C09104=1083.257,-6.050,442.174,174.206,19.488,153.253
C09105=1083.262,-5.800,442.160,174.207,19.490,153.253
C09106=1083.268,-5.551,442.147,174.208,19.492,153.254
C09107=1083.274,-5.301,442.133,174.210,19.495,153.254
C09108=1083.280,-5.052,442.120,174.212,19.496,153.254
C09109=1083.285,-4.803,442.106,174.213,19.498,153.254
C09110=1083.292,-4.553,442.092,174.214,19.500,153.254
C09111=1083.298,-4.303,442.078,174.216,19.503,153.254
C09112=1083.303,-4.053,442.064,174.218,19.504,153.254
C09113=1083.309,-3.804,442.051,174.219,19.506,153.254
C09114=1083.315,-3.555,442.037,174.220,19.508,153.255
C09115=1083.321,-3.305,442.024,174.222,19.510,153.255
C09116=1083.327,-3.055,442.010,174.224,19.512,153.255
C09117=1083.333,-2.805,441.996,174.225,19.514,153.255
C09118=1083.338,-2.556,441.982,174.226,19.516,153.255
C09119=1083.344,-2.307,441.969,174.228,19.519,153.255
C09120=1083.350,-2.057,441.955,174.229,19.521,153.255
C09121=1083.355,-1.807,441.941,174.231,19.523,153.256
C09122=1083.361,-1.558,441.927,174.232,19.524,153.256
C09123=1083.368,-1.282,441.912,174.234,19.527,153.256
C09124=1083.374,-1.007,441.897,174.235,19.529,153.256
C09125=1083.380,-0.732,441.882,174.237,19.532,153.256
C09126=1083.387,-0.457,441.866,174.238,19.534,153.256
C09127=1083.392,-0.207,441.852,174.241,19.536,153.256
C09128=1083.398,0.043,441.838,174.242,19.538,153.257
C09129=1083.403,0.292,441.824,174.243,19.540,153.257
C09130=1083.410,0.541,441.811,174.244,19.542,153.257
C09131=1083.416,0.792,441.796,174.247,19.545,153.257
C09132=1083.421,1.041,441.783,174.248,19.547,153.257
C09133=1083.427,1.290,441.768,174.249,19.548,153.257
C09134=1083.432,1.540,441.754,174.250,19.550,153.257
C09135=1083.439,1.789,441.741,174.253,19.553,153.258
C09136=1083.445,2.039,441.727,174.254,19.555,153.258
C09137=1083.450,2.289,441.713,174.255,19.557,153.258
C09138=1083.456,2.538,441.699,174.256,19.559,153.258
C09139=1083.461,2.787,441.684,174.259,19.561,153.258
C09140=1083.467,3.037,441.670,174.260,19.563,153.258
C09141=1083.474,3.287,441.657,174.261,19.565,153.258
C09142=1083.479,3.537,441.643,174.262,19.567,153.259
C09143=1083.485,3.785,441.628,174.264,19.569,153.259
C09144=1083.490,4.035,441.615,174.266,19.571,153.259
C09145=1083.496,4.285,441.600,174.267,19.573,153.259
C09146=1083.502,4.535,441.586,174.268,19.575,153.259
C09147=1083.508,4.784,441.572,174.270,19.577,153.259
C09148=1083.514,5.033,441.559,174.272,19.579,153.259
C09149=1083.520,5.283,441.544,174.273,19.581,153.260
C09150=1083.525,5.533,441.531,174.274,19.583,153.260
C09151=1083.531,5.782,441.516,174.276,19.585,153.260
C09152=1083.537,6.032,441.502,174.278,19.587,153.260
C09153=1083.543,6.282,441.488,174.279,19.589,153.260
C09154=1083.549,6.531,441.473,174.281,19.592,153.260
C09155=1083.554,6.780,441.459,174.282,19.594,153.261
C09156=1083.561,7.030,441.446,174.284,19.595,153.261
C09157=1083.567,7.279,441.431,174.285,19.597,153.261
C09158=1083.572,7.529,441.417,174.287,19.600,153.261
C09159=1083.578,7.778,441.403,174.288,19.602,153.261
C09160=1083.584,8.028,441.388,174.289,19.604,153.261
C09161=1083.589,8.278,441.375,174.291,19.606,153.261
C09162=1083.595,8.527,441.360,174.293,19.608,153.261
C09163=1083.601,8.777,441.346,174.294,19.610,153.262
C09164=1083.607,9.026,441.332,174.295,19.612,153.262
C09165=1083.613,9.275,441.317,174.298,19.615,153.262
C09166=1083.619,9.526,441.303,174.299,19.616,153.262
C09167=1083.625,9.774,441.289,174.300,19.618,153.262
C09168=1083.631,10.024,441.275,174.301,19.620,153.262
C09169=1083.637,10.274,441.260,174.304,19.623,153.262
C09170=1083.643,10.523,441.246,174.305,19.625,153.263
C09171=1083.649,10.773,441.232,174.306,19.626,153.263
C09172=1083.654,11.022,441.218,174.308,19.628,153.263
C09173=1083.660,11.272,441.204,174.310,19.631,153.263
C09174=1083.666,11.522,441.189,174.311,19.633,153.263
C09175=1083.672,11.771,441.175,174.312,19.635,153.263
C09176=1083.678,12.020,441.160,174.314,19.637,153.263
C09177=1083.684,12.270,441.146,174.316,19.639,153.263
C09178=1083.689,12.519,441.132,174.317,19.641,153.264
C09179=1083.695,12.770,441.117,174.318,19.643,153.264
C09180=1083.701,13.019,441.103,174.320,19.645,153.264
C09181=1083.707,13.268,441.089,174.322,19.647,153.264
C09182=1083.713,13.518,441.074,174.323,19.649,153.264
C09183=1083.719,13.767,441.059,174.325,19.651,153.264
C09184=1083.725,14.017,441.045,174.326,19.653,153.264
C09185=1083.731,14.266,441.031,174.328,19.655,153.265
C09186=1083.736,14.516,441.017,174.329,19.657,153.265
C09187=1083.744,14.793,441.000,174.331,19.659,153.265
C09188=1083.749,15.071,440.984,174.332,19.661,153.265
C09189=1083.756,15.348,440.968,174.334,19.664,153.265
C09190=1083.763,15.625,440.952,174.336,19.666,153.265
C09191=1083.768,15.874,440.937,174.338,19.668,153.265
C09192=1083.774,16.125,440.923,174.339,19.670,153.266
C09193=1083.780,16.373,440.908,174.340,19.672,153.266
C09194=1083.786,16.623,440.894,174.342,19.675,153.266
C09195=1083.791,16.873,440.880,174.344,19.676,153.266
C09196=1083.797,17.122,440.865,174.345,19.678,153.266
C09197=1083.803,17.372,440.850,174.347,19.681,153.266
C09198=1083.808,17.621,440.836,174.348,19.683,153.267
C09199=1083.815,17.871,440.821,174.350,19.685,153.267
C09200=1083.820,18.120,440.806,174.352,19.687,153.267
C09201=1083.827,18.370,440.792,174.353,19.689,153.267
C09202=1083.832,18.619,440.777,174.354,19.691,153.267
C09203=1083.837,18.868,440.762,174.356,19.693,153.267
C09204=1083.844,19.118,440.747,174.358,19.695,153.267
C09205=1083.849,19.368,440.733,174.359,19.697,153.268
C09206=1083.856,19.617,440.718,174.360,19.699,153.268
C09207=1083.861,19.866,440.704,174.362,19.701,153.268
C09208=1083.867,20.117,440.689,174.364,19.703,153.268
C09209=1083.872,20.366,440.674,174.365,19.706,153.268
C09210=1083.879,20.615,440.659,174.367,19.708,153.268
C09211=1083.885,20.864,440.645,174.368,19.710,153.268
C09212=1083.889,21.114,440.630,174.370,19.712,153.268
C09213=1083.896,21.364,440.615,174.371,19.714,153.269
C09214=1083.902,21.613,440.601,174.373,19.716,153.269
C09215=1083.907,21.863,440.585,174.374,19.718,153.269
C09216=1083.913,22.112,440.571,174.376,19.720,153.269
C09217=1083.919,22.362,440.557,174.378,19.723,153.269
C09218=1083.924,22.611,440.541,174.379,19.725,153.269
C09219=1083.930,22.861,440.526,174.380,19.726,153.269
C09220=1083.936,23.110,440.512,174.382,19.729,153.270
C09221=1083.942,23.360,440.496,174.384,19.731,153.270
C09222=1083.948,23.609,440.482,174.385,19.733,153.270
C09223=1083.954,23.859,440.467,174.387,19.735,153.270
C09224=1083.959,24.108,440.452,174.389,19.737,153.270
C09225=1083.965,24.358,440.437,174.390,19.739,153.270
C09226=1083.971,24.607,440.423,174.392,19.741,153.270
C09227=1083.977,24.857,440.407,174.393,19.743,153.271
C09228=1083.982,25.106,440.393,174.394,19.745,153.271
C09229=1083.989,25.356,440.378,174.396,19.748,153.271
C09230=1083.994,25.605,440.363,174.398,19.749,153.271
C09231=1084.000,25.854,440.348,174.399,19.751,153.271
C09232=1084.006,26.103,440.333,174.400,19.753,153.271
C09233=1084.012,26.353,440.317,174.403,19.756,153.271
C09234=1084.017,26.603,440.304,174.404,19.758,153.272
C09235=1084.024,26.853,440.289,174.405,19.759,153.272
C09236=1084.029,27.102,440.274,174.407,19.762,153.272
C09237=1084.035,27.352,440.259,174.409,19.764,153.272
C09238=1084.040,27.601,440.243,174.410,19.766,153.272
C09239=1084.046,27.850,440.228,174.412,19.768,153.272
C09240=1084.052,28.100,440.213,174.413,19.770,153.272
C09241=1084.058,28.349,440.198,174.415,19.772,153.273
C09242=1084.064,28.599,440.183,174.417,19.774,153.273
C09243=1084.069,28.848,440.168,174.418,19.776,153.273
C09244=1084.076,29.098,440.153,174.419,19.778,153.273
C09245=1084.081,29.347,440.138,174.422,19.780,153.273
C09246=1084.087,29.597,440.123,174.423,19.782,153.273
C09247=1084.092,29.846,440.108,174.424,19.784,153.273
C09248=1084.098,30.096,440.093,174.426,19.787,153.274
C09249=1084.104,30.345,440.077,174.427,19.789,153.274
C09250=1084.109,30.594,440.062,174.429,19.791,153.274
C09251=1084.116,30.874,440.045,174.431,19.793,153.274
C09252=1084.123,31.152,440.028,174.433,19.796,153.274
C09253=1084.128,31.431,440.011,174.434,19.798,153.274
C09254=1084.135,31.710,439.995,174.436,19.800,153.275
C09255=1084.141,31.959,439.978,174.437,19.802,153.275
C09256=1084.147,32.208,439.964,174.440,19.804,153.275
C09257=1084.153,32.458,439.948,174.441,19.806,153.275
C09258=1084.158,32.707,439.934,174.442,19.808,153.275
C09259=1084.164,32.957,439.918,174.444,19.811,153.275
C09260=1084.170,33.207,439.903,174.446,19.813,153.275
C09261=1084.176,33.456,439.888,174.447,19.814,153.275
C09262=1084.181,33.705,439.872,174.449,19.817,153.276
C09263=1084.187,33.954,439.857,174.450,19.819,153.276
C09264=1084.193,34.204,439.842,174.452,19.821,153.276
C09265=1084.199,34.454,439.827,174.454,19.823,153.276
C09266=1084.204,34.703,439.811,174.455,19.825,153.276
C09267=1084.211,34.952,439.796,174.456,19.827,153.276
C09268=1084.217,35.202,439.780,174.459,19.829,153.276
C09269=1084.222,35.451,439.765,174.460,19.831,153.277
C09270=1084.228,35.701,439.750,174.461,19.833,153.277
C09271=1084.234,35.951,439.735,174.463,19.835,153.277
C09272=1084.239,36.200,439.719,174.465,19.837,153.277
C09273=1084.245,36.449,439.704,174.466,19.839,153.277
C09274=1084.251,36.699,439.688,174.468,19.842,153.277
C09275=1084.257,36.948,439.673,174.469,19.843,153.277
C09276=1084.263,37.198,439.657,174.471,19.845,153.277
C09277=1084.268,37.448,439.642,174.473,19.848,153.278
C09278=1084.274,37.697,439.627,174.474,19.850,153.278
C09279=1084.280,37.946,439.611,174.476,19.852,153.278
C09280=1084.286,38.196,439.595,174.478,19.854,153.278
C09281=1084.291,38.445,439.580,174.479,19.856,153.278
C09282=1084.298,38.694,439.565,174.481,19.858,153.278
C09283=1084.303,38.944,439.549,174.482,19.860,153.278
C09284=1084.308,39.193,439.534,174.484,19.862,153.279
C09285=1084.314,39.443,439.518,174.486,19.864,153.279
C09286=1084.321,39.692,439.503,174.487,19.866,153.279
C09287=1084.326,39.942,439.487,174.488,19.868,153.279
C09288=1084.332,40.191,439.471,174.490,19.871,153.279
C09289=1084.337,40.441,439.456,174.492,19.872,153.279
C09290=1084.343,40.690,439.440,174.494,19.875,153.279
C09291=1084.349,40.939,439.425,174.495,19.877,153.280
C09292=1084.355,41.189,439.409,174.497,19.879,153.280
C09293=1084.360,41.438,439.393,174.499,19.881,153.280
C09294=1084.366,41.688,439.378,174.500,19.883,153.280
C09295=1084.372,41.937,439.362,174.501,19.885,153.280
C09296=1084.378,42.187,439.347,174.503,19.887,153.280
C09297=1084.383,42.436,439.331,174.505,19.889,153.280
C09298=1084.389,42.686,439.315,174.506,19.891,153.280
C09299=1084.395,42.936,439.300,174.508,19.893,153.281
C09300=1084.400,43.184,439.284,174.510,19.895,153.281
C09301=1084.406,43.434,439.268,174.512,19.898,153.281
C09302=1084.412,43.683,439.253,174.513,19.899,153.281
C09303=1084.418,43.933,439.237,174.514,19.901,153.281
C09304=1084.423,44.182,439.221,174.516,19.904,153.281
C09305=1084.429,44.432,439.206,174.518,19.906,153.281
C09306=1084.435,44.681,439.189,174.519,19.908,153.282
C09307=1084.440,44.930,439.174,174.521,19.910,153.282
C09308=1084.446,45.180,439.158,174.523,19.912,153.282
C09309=1084.452,45.430,439.142,174.525,19.914,153.282
C09310=1084.457,45.679,439.126,174.526,19.916,153.282
C09311=1084.463,45.928,439.110,174.527,19.918,153.282
C09312=1084.468,46.178,439.095,174.529,19.921,153.282
C09313=1084.474,46.427,439.078,174.531,19.922,153.282
C09314=1084.479,46.677,439.062,174.533,19.925,153.283
C09315=1084.486,46.955,439.045,174.534,19.927,153.283
C09316=1084.492,47.234,439.027,174.536,19.929,153.283
C09317=1084.499,47.513,439.010,174.538,19.932,153.283
C09318=1084.505,47.791,438.992,174.540,19.934,153.283
C09319=1084.511,48.041,438.976,174.542,19.936,153.283
C09320=1084.516,48.291,438.960,174.543,19.938,153.284
C09321=1084.522,48.540,438.944,174.544,19.940,153.284
C09322=1084.527,48.789,438.928,174.547,19.942,153.284
C09323=1084.533,49.039,438.912,174.548,19.944,153.284
C09324=1084.538,49.288,438.896,174.550,19.946,153.284
C09325=1084.544,49.538,438.879,174.551,19.948,153.284
C09326=1084.550,49.788,438.864,174.553,19.950,153.284
C09327=1084.555,50.036,438.848,174.555,19.952,153.284
C09328=1084.561,50.286,438.832,174.556,19.954,153.285
C09329=1084.567,50.535,438.815,174.558,19.956,153.285
C09330=1084.573,50.785,438.800,174.560,19.958,153.285
C09331=1084.579,51.034,438.784,174.561,19.960,153.285
C09332=1084.584,51.283,438.768,174.563,19.963,153.285
C09333=1084.590,51.533,438.752,174.564,19.964,153.285
C09334=1084.596,51.782,438.736,174.567,19.967,153.285
C09335=1084.602,52.032,438.720,174.568,19.969,153.285
C09336=1084.607,52.281,438.703,174.569,19.971,153.286
C09337=1084.613,52.531,438.687,174.571,19.973,153.286
C09338=1084.618,52.780,438.671,174.573,19.975,153.286
C09339=1084.624,53.029,438.655,174.575,19.977,153.286
C09340=1084.630,53.279,438.639,174.576,19.979,153.286
C09341=1084.636,53.528,438.623,174.577,19.981,153.286
C09342=1084.641,53.778,438.607,174.580,19.983,153.286
C09343=1084.647,54.027,438.591,174.581,19.985,153.286
C09344=1084.653,54.277,438.574,174.583,19.987,153.287
C09345=1084.659,54.526,438.558,174.584,19.989,153.287
C09346=1084.664,54.775,438.542,174.586,19.991,153.287
C09347=1084.670,55.024,438.526,174.588,19.993,153.287
C09348=1084.676,55.274,438.509,174.589,19.995,153.287
C09349=1084.681,55.524,438.494,174.592,19.997,153.287
C09350=1084.687,55.773,438.477,174.593,19.999,153.287
C09351=1084.693,56.023,438.461,174.594,20.001,153.287
C09352=1084.699,56.272,438.444,174.597,20.003,153.287
C09353=1084.704,56.521,438.428,174.598,20.005,153.288
C09354=1084.710,56.771,438.412,174.600,20.008,153.288
C09355=1084.716,57.020,438.396,174.601,20.009,153.288
C09356=1084.722,57.269,438.379,174.603,20.011,153.288
C09357=1084.728,57.519,438.362,174.605,20.014,153.288
C09358=1084.733,57.768,438.346,174.606,20.015,153.288
C09359=1084.739,58.017,438.330,174.608,20.018,153.288
C09360=1084.745,58.266,438.314,174.610,20.019,153.288
C09361=1084.751,58.516,438.298,174.612,20.022,153.289
C09362=1084.757,58.765,438.282,174.613,20.024,153.289
C09363=1084.762,59.015,438.265,174.615,20.025,153.289
C09364=1084.768,59.264,438.248,174.617,20.028,153.289
C09365=1084.774,59.513,438.232,174.618,20.029,153.289
C09366=1084.780,59.763,438.216,174.620,20.031,153.289
C09367=1084.786,60.012,438.200,174.622,20.033,153.289
C09368=1084.791,60.262,438.183,174.624,20.035,153.289
C09369=1084.797,60.511,438.167,174.625,20.037,153.289
C09370=1084.803,60.761,438.150,174.627,20.039,153.289
C09371=1084.809,61.010,438.134,174.629,20.041,153.290
C09372=1084.814,61.260,438.117,174.630,20.043,153.290
C09373=1084.820,61.509,438.101,174.632,20.045,153.290
C09374=1084.826,61.758,438.085,174.634,20.047,153.290
C09375=1084.832,62.008,438.068,174.635,20.049,153.290
C09376=1084.838,62.257,438.052,174.637,20.051,153.290
C09377=1084.843,62.507,438.035,174.639,20.053,153.290
C09378=1084.850,62.757,438.019,174.641,20.055,153.290
C09379=1084.856,63.034,438.000,174.642,20.057,153.290
C09380=1084.862,63.313,437.982,174.644,20.059,153.291
C09381=1084.869,63.591,437.963,174.647,20.062,153.291
C09382=1084.876,63.870,437.945,174.649,20.064,153.291
C09383=1084.881,64.120,437.928,174.650,20.066,153.291
C09384=1084.887,64.369,437.912,174.652,20.068,153.291
C09385=1084.893,64.618,437.895,174.654,20.070,153.291
C09386=1084.898,64.867,437.878,174.655,20.072,153.291
C09387=1084.904,65.117,437.862,174.657,20.074,153.291
C09388=1084.909,65.366,437.845,174.659,20.076,153.291
C09389=1084.916,65.616,437.829,174.661,20.078,153.292
C09390=1084.922,65.865,437.812,174.662,20.080,153.292
C09391=1084.927,66.115,437.795,174.664,20.082,153.292
C09392=1084.933,66.364,437.778,174.666,20.084,153.292
C09393=1084.939,66.614,437.762,174.667,20.086,153.292
C09394=1084.945,66.863,437.745,174.669,20.087,153.292
C09395=1084.950,67.112,437.728,174.671,20.089,153.292
C09396=1084.956,67.362,437.712,174.673,20.092,153.292
C09397=1084.961,67.611,437.695,174.674,20.093,153.292
C09398=1084.967,67.860,437.678,174.676,20.096,153.292
C09399=1084.973,68.110,437.661,174.678,20.097,153.293
C09400=1084.979,68.359,437.645,174.680,20.100,153.293
C09401=1084.984,68.608,437.627,174.682,20.101,153.293
C09402=1084.990,68.857,437.611,174.684,20.104,153.293
C09403=1084.995,69.107,437.594,174.685,20.105,153.293
C09404=1085.002,69.356,437.577,174.686,20.107,153.293
C09405=1085.007,69.606,437.560,174.689,20.109,153.293
C09406=1085.013,69.855,437.543,174.690,20.111,153.293
C09407=1085.019,70.105,437.526,174.692,20.114,153.293
C09408=1085.025,70.354,437.510,174.694,20.115,153.293
C09409=1085.030,70.604,437.493,174.696,20.118,153.294
C09410=1085.036,70.853,437.475,174.697,20.119,153.294
C09411=1085.042,71.102,437.459,174.699,20.122,153.294
C09412=1085.047,71.352,437.442,174.701,20.123,153.294
C09413=1085.053,71.600,437.425,174.703,20.126,153.294
C09414=1085.058,71.850,437.408,174.704,20.127,153.294
C09415=1085.064,72.099,437.391,174.706,20.129,153.294
C09416=1085.070,72.349,437.374,174.708,20.131,153.294
C09417=1085.076,72.598,437.357,174.709,20.133,153.294
C09418=1085.081,72.848,437.340,174.712,20.135,153.294
C09419=1085.087,73.097,437.323,174.713,20.137,153.295
C09420=1085.092,73.346,437.306,174.715,20.139,153.295
C09421=1085.098,73.596,437.289,174.717,20.141,153.295
C09422=1085.104,73.845,437.272,174.719,20.143,153.295
C09423=1085.109,74.094,437.255,174.720,20.145,153.295
C09424=1085.115,74.344,437.237,174.722,20.147,153.295
C09425=1085.121,74.593,437.221,174.724,20.149,153.295
C09426=1085.127,74.842,437.203,174.726,20.151,153.295
C09427=1085.132,75.092,437.187,174.727,20.153,153.295
C09428=1085.138,75.341,437.170,174.730,20.155,153.295
C09429=1085.144,75.590,437.152,174.731,20.157,153.295
C09430=1085.150,75.840,437.135,174.733,20.159,153.295
C09431=1085.155,76.089,437.117,174.735,20.161,153.296
C09432=1085.161,76.339,437.101,174.737,20.163,153.296
C09433=1085.167,76.588,437.083,174.738,20.165,153.296
C09434=1085.172,76.837,437.067,174.740,20.166,153.296
C09435=1085.179,77.087,437.049,174.742,20.169,153.296
C09436=1085.184,77.336,437.032,174.743,20.170,153.296
C09437=1085.189,77.585,437.015,174.745,20.173,153.296
C09438=1085.195,77.834,436.997,174.747,20.174,153.296
C09439=1085.201,78.084,436.981,174.749,20.176,153.296
C09440=1085.207,78.333,436.963,174.751,20.178,153.296
C09441=1085.212,78.583,436.946,174.753,20.180,153.296
C09442=1085.218,78.832,436.929,174.754,20.182,153.297
C09443=1085.224,79.110,436.910,174.757,20.184,153.297
C09444=1085.231,79.389,436.890,174.759,20.186,153.297
C09445=1085.237,79.667,436.870,174.761,20.189,153.297
C09446=1085.243,79.945,436.851,174.762,20.190,153.297
C09447=1085.248,80.195,436.834,174.764,20.193,153.297
C09448=1085.254,80.445,436.816,174.766,20.194,153.297
C09449=1085.260,80.694,436.799,174.768,20.197,153.297
C09450=1085.266,80.943,436.782,174.769,20.198,153.297
C09451=1085.271,81.192,436.765,174.772,20.201,153.297
C09452=1085.277,81.441,436.747,174.773,20.202,153.298
C09453=1085.283,81.691,436.729,174.775,20.205,153.298
C09454=1085.288,81.941,436.712,174.777,20.206,153.298
C09455=1085.294,82.190,436.695,174.779,20.208,153.298
C09456=1085.299,82.439,436.677,174.780,20.210,153.298
C09457=1085.305,82.688,436.659,174.783,20.212,153.298
C09458=1085.311,82.937,436.642,174.784,20.214,153.298
C09459=1085.316,83.187,436.625,174.786,20.216,153.298
C09460=1085.322,83.436,436.607,174.788,20.218,153.298
C09461=1085.328,83.686,436.589,174.790,20.220,153.298
C09462=1085.333,83.935,436.572,174.791,20.221,153.298
C09463=1085.339,84.184,436.554,174.794,20.224,153.298
C09464=1085.344,84.434,436.537,174.795,20.225,153.299
C09465=1085.350,84.683,436.519,174.797,20.228,153.299
C09466=1085.356,84.932,436.502,174.799,20.229,153.299
C09467=1085.361,85.181,436.484,174.801,20.231,153.299
C09468=1085.367,85.431,436.466,174.802,20.233,153.299
C09469=1085.373,85.680,436.449,174.805,20.235,153.299
C09470=1085.379,85.929,436.432,174.807,20.237,153.299
C09471=1085.385,86.179,436.414,174.808,20.239,153.299
C09472=1085.391,86.428,436.396,174.811,20.241,153.299
C09473=1085.396,86.677,436.379,174.812,20.242,153.299
C09474=1085.402,86.927,436.362,174.814,20.245,153.299
C09475=1085.408,87.176,436.344,174.816,20.246,153.299
C09476=1085.413,87.425,436.326,174.818,20.248,153.299
C09477=1085.419,87.675,436.308,174.819,20.250,153.300
C09478=1085.425,87.924,436.291,174.822,20.252,153.300
C09479=1085.430,88.173,436.273,174.823,20.254,153.300
C09480=1085.436,88.423,436.255,174.825,20.256,153.300
C09481=1085.442,88.672,436.238,174.827,20.258,153.300
C09482=1085.447,88.921,436.220,174.829,20.260,153.300
C09483=1085.453,89.171,436.202,174.831,20.261,153.300
C09484=1085.458,89.420,436.184,174.833,20.264,153.300
C09485=1085.464,89.669,436.167,174.834,20.265,153.300
C09486=1085.470,89.919,436.149,174.837,20.267,153.300
C09487=1085.475,90.168,436.131,174.838,20.269,153.300
C09488=1085.482,90.418,436.113,174.840,20.271,153.300
C09489=1085.487,90.667,436.096,174.842,20.272,153.300
C09490=1085.493,90.916,436.077,174.844,20.274,153.300
C09491=1085.499,91.165,436.059,174.845,20.276,153.300
C09492=1085.504,91.414,436.042,174.848,20.278,153.300
C09493=1085.511,91.663,436.024,174.850,20.280,153.300
C09494=1085.515,91.913,436.006,174.851,20.282,153.301
C09495=1085.521,92.162,435.988,174.854,20.284,153.301
C09496=1085.527,92.412,435.970,174.855,20.286,153.301
C09497=1085.533,92.661,435.953,174.857,20.288,153.301
C09498=1085.537,92.910,435.935,174.859,20.290,153.301
C09499=1085.544,93.159,435.916,174.861,20.292,153.301
C09500=1085.549,93.408,435.898,174.863,20.293,153.301
C09501=1085.555,93.658,435.880,174.865,20.296,153.301
C09502=1085.560,93.907,435.862,174.866,20.297,153.301
C09503=1085.566,94.156,435.845,174.869,20.299,153.301
C09504=1085.572,94.406,435.827,174.870,20.301,153.301
C09505=1085.578,94.654,435.808,174.872,20.303,153.301
C09506=1085.583,94.905,435.790,174.875,20.305,153.301
C09507=1085.589,95.183,435.770,174.876,20.306,153.301
C09508=1085.595,95.461,435.750,174.878,20.309,153.302
C09509=1085.602,95.740,435.730,174.881,20.311,153.302
C09510=1085.608,96.018,435.710,174.883,20.313,153.302
C09511=1085.614,96.267,435.691,174.885,20.315,153.302
C09512=1085.620,96.517,435.674,174.887,20.317,153.302
C09513=1085.625,96.767,435.655,174.889,20.319,153.302
C09514=1085.631,97.016,435.637,174.890,20.321,153.302
C09515=1085.637,97.265,435.619,174.893,20.323,153.302
C09516=1085.643,97.514,435.601,174.894,20.324,153.302
C09517=1085.647,97.763,435.583,174.896,20.326,153.302
C09518=1085.654,98.012,435.564,174.898,20.327,153.302
C09519=1085.659,98.261,435.547,174.900,20.329,153.302
C09520=1085.665,98.511,435.528,174.902,20.332,153.302
C09521=1085.671,98.760,435.510,174.904,20.333,153.302
C09522=1085.677,99.010,435.492,174.906,20.335,153.302
C09523=1085.681,99.259,435.474,174.908,20.337,153.302
C09524=1085.688,99.508,435.455,174.910,20.339,153.302
C09525=1085.693,99.757,435.438,174.912,20.340,153.302
C09526=1085.699,100.006,435.419,174.914,20.343,153.302
C09527=1085.705,100.256,435.401,174.915,20.344,153.303
C09528=1085.711,100.505,435.383,174.918,20.346,153.303
C09529=1085.716,100.755,435.364,174.920,20.348,153.303
C09530=1085.722,101.004,435.346,174.921,20.349,153.303
C09531=1085.728,101.253,435.328,174.924,20.351,153.303
C09532=1085.733,101.502,435.309,174.925,20.353,153.303
C09533=1085.740,101.751,435.291,174.927,20.355,153.303
C09534=1085.744,102.001,435.273,174.929,20.357,153.303
C09535=1085.750,102.250,435.255,174.931,20.359,153.303
C09536=1085.756,102.499,435.236,174.934,20.361,153.303
C09537=1085.761,102.749,435.217,174.935,20.362,153.303
C09538=1085.767,102.998,435.199,174.937,20.365,153.303
C09539=1085.772,103.248,435.180,174.939,20.366,153.303
C09540=1085.778,103.496,435.162,174.941,20.368,153.303
C09541=1085.783,103.746,435.144,174.943,20.370,153.303
C09542=1085.789,103.995,435.125,174.945,20.371,153.303
C09543=1085.795,104.244,435.106,174.947,20.373,153.303
C09544=1085.800,104.493,435.089,174.949,20.375,153.303
C09545=1085.806,104.742,435.069,174.951,20.377,153.303
C09546=1085.812,104.992,435.051,174.952,20.379,153.303
C09547=1085.817,105.241,435.033,174.955,20.381,153.303
C09548=1085.823,105.491,435.014,174.957,20.383,153.303
C09549=1085.828,105.739,434.996,174.959,20.384,153.303
C09550=1085.834,105.989,434.976,174.961,20.386,153.303
C09551=1085.840,106.238,434.959,174.963,20.388,153.303
C09552=1085.845,106.487,434.940,174.965,20.390,153.303
C09553=1085.851,106.737,434.922,174.967,20.392,153.303
C09554=1085.857,106.986,434.903,174.969,20.393,153.304
C09555=1085.862,107.235,434.884,174.971,20.395,153.304
C09556=1085.868,107.484,434.866,174.972,20.397,153.304
C09557=1085.873,107.734,434.847,174.975,20.399,153.304
C09558=1085.880,107.983,434.828,174.977,20.401,153.304
C09559=1085.885,108.232,434.810,174.979,20.402,153.304
C09560=1085.890,108.482,434.791,174.981,20.404,153.304
C09561=1085.897,108.731,434.772,174.982,20.406,153.304
C09562=1085.902,108.979,434.753,174.985,20.408,153.304
C09563=1085.908,109.229,434.735,174.987,20.410,153.304
C09564=1085.913,109.478,434.716,174.989,20.411,153.304
C09565=1085.919,109.727,434.697,174.991,20.413,153.304
C09566=1085.925,109.976,434.678,174.993,20.414,153.304
C09567=1085.930,110.226,434.660,174.995,20.416,153.304
C09568=1085.936,110.475,434.641,174.997,20.418,153.304
C09569=1085.942,110.724,434.622,174.999,20.420,153.304
C09570=1085.948,110.974,434.603,175.001,20.422,153.304
C09571=1085.953,111.252,434.582,175.003,20.424,153.304
C09572=1085.960,111.531,434.562,175.006,20.426,153.304
C09573=1085.967,111.810,434.541,175.008,20.428,153.304
C09574=1085.973,112.088,434.520,175.010,20.429,153.304
C09575=1085.978,112.337,434.501,175.012,20.431,153.304
C09576=1085.984,112.586,434.482,175.014,20.433,153.304
C09577=1085.990,112.836,434.463,175.016,20.434,153.304
C09578=1085.995,113.084,434.444,175.018,20.436,153.304
C09579=1086.001,113.334,434.425,175.021,20.438,153.304
C09580=1086.007,113.583,434.406,175.022,20.440,153.304
C09581=1086.012,113.832,434.387,175.025,20.442,153.304
C09582=1086.018,114.082,434.369,175.026,20.443,153.304
C09583=1086.023,114.331,434.350,175.028,20.445,153.304
C09584=1086.029,114.580,434.331,175.031,20.447,153.304
C09585=1086.034,114.829,434.311,175.032,20.449,153.304
C09586=1086.040,115.079,434.292,175.035,20.451,153.304
C09587=1086.045,115.328,434.273,175.037,20.452,153.304
C09588=1086.051,115.577,434.255,175.038,20.454,153.304
C09589=1086.057,115.826,434.235,175.041,20.456,153.305
C09590=1086.062,116.075,434.217,175.042,20.458,153.305
C09591=1086.068,116.324,434.197,175.044,20.460,153.305
C09592=1086.074,116.574,434.178,175.047,20.462,153.305
C09593=1086.079,116.823,434.159,175.048,20.463,153.305
C09594=1086.084,117.072,434.140,175.051,20.465,153.305
C09595=1086.090,117.321,434.121,175.053,20.467,153.305
C09596=1086.096,117.571,434.101,175.055,20.469,153.305
C09597=1086.101,117.819,434.083,175.057,20.471,153.305
C09598=1086.106,118.069,434.063,175.059,20.472,153.305
C09599=1086.112,118.318,434.044,175.061,20.473,153.305
C09600=1086.118,118.568,434.025,175.063,20.475,153.305
C09601=1086.123,118.817,434.006,175.066,20.477,153.305
C09602=1086.129,119.066,433.987,175.067,20.479,153.305
C09603=1086.134,119.315,433.968,175.070,20.481,153.305
C09604=1086.140,119.564,433.948,175.071,20.482,153.305
C09605=1086.145,119.813,433.929,175.073,20.484,153.305
C09606=1086.151,120.062,433.909,175.076,20.486,153.305
C09607=1086.157,120.312,433.890,175.077,20.488,153.305
C09608=1086.162,120.561,433.871,175.080,20.489,153.305
C09609=1086.168,120.810,433.852,175.082,20.491,153.305
C09610=1086.173,121.059,433.833,175.084,20.493,153.305
C09611=1086.179,121.308,433.813,175.086,20.495,153.305
C09612=1086.185,121.558,433.794,175.088,20.497,153.305
C09613=1086.191,121.807,433.774,175.090,20.498,153.305
C09614=1086.196,122.056,433.755,175.092,20.500,153.305
C09615=1086.201,122.305,433.736,175.095,20.502,153.305
C09616=1086.207,122.555,433.717,175.096,20.503,153.305
C09617=1086.212,122.804,433.696,175.099,20.505,153.305
C09618=1086.218,123.053,433.677,175.101,20.507,153.305
C09619=1086.223,123.302,433.658,175.102,20.508,153.305
C09620=1086.229,123.551,433.639,175.105,20.510,153.305
C09621=1086.235,123.800,433.619,175.107,20.512,153.305
C09622=1086.240,124.050,433.600,175.109,20.513,153.305
C09623=1086.246,124.299,433.581,175.111,20.515,153.305
C09624=1086.252,124.548,433.561,175.114,20.517,153.305
C09625=1086.258,124.797,433.541,175.115,20.519,153.305
C09626=1086.263,125.046,433.523,175.118,20.520,153.305
C09627=1086.269,125.295,433.503,175.120,20.522,153.305
C09628=1086.275,125.544,433.483,175.122,20.523,153.305
C09629=1086.280,125.794,433.464,175.124,20.525,153.305
C09630=1086.286,126.043,433.444,175.127,20.527,153.305
C09631=1086.291,126.292,433.424,175.128,20.528,153.305
C09632=1086.297,126.542,433.405,175.130,20.530,153.305
C09633=1086.303,126.791,433.385,175.133,20.532,153.305
C09634=1086.309,127.040,433.366,175.134,20.533,153.305
C09635=1086.315,127.318,433.344,175.137,20.535,153.305
C09636=1086.321,127.597,433.322,175.139,20.537,153.305
C09637=1086.328,127.875,433.300,175.142,20.539,153.305
C09638=1086.334,128.154,433.279,175.144,20.541,153.305
C09639=1086.340,128.403,433.259,175.147,20.542,153.305
C09640=1086.345,128.652,433.240,175.149,20.544,153.305
C09641=1086.351,128.901,433.219,175.151,20.546,153.305
C09642=1086.356,129.151,433.200,175.153,20.548,153.305
C09643=1086.362,129.400,433.180,175.155,20.549,153.305
C09644=1086.368,129.649,433.161,175.158,20.551,153.305
C09645=1086.374,129.898,433.141,175.159,20.553,153.305
C09646=1086.380,130.147,433.121,175.162,20.554,153.305
C09647=1086.386,130.396,433.101,175.164,20.556,153.305
C09648=1086.391,130.646,433.082,175.166,20.557,153.305
C09649=1086.397,130.895,433.062,175.168,20.559,153.305
C09650=1086.402,131.144,433.042,175.171,20.561,153.305
C09651=1086.408,131.393,433.022,175.173,20.563,153.305
C09652=1086.414,131.642,433.003,175.175,20.564,153.304
C09653=1086.419,131.892,432.983,175.177,20.566,153.305
C09654=1086.425,132.140,432.963,175.180,20.567,153.304
C09655=1086.431,132.390,432.943,175.181,20.568,153.304
C09656=1086.437,132.639,432.923,175.184,20.570,153.304
C09657=1086.442,132.888,432.904,175.186,20.572,153.304
C09658=1086.448,133.137,432.884,175.188,20.574,153.304
C09659=1086.453,133.386,432.863,175.190,20.575,153.304
C09660=1086.458,133.635,432.844,175.192,20.577,153.304
C09661=1086.464,133.884,432.824,175.195,20.579,153.304
C09662=1086.470,134.133,432.804,175.196,20.580,153.304
C09663=1086.475,134.382,432.784,175.199,20.582,153.304
C09664=1086.480,134.631,432.764,175.201,20.584,153.304
C09665=1086.486,134.880,432.744,175.204,20.585,153.304
C09666=1086.492,135.130,432.725,175.205,20.587,153.304
C09667=1086.497,135.379,432.704,175.208,20.589,153.304
C09668=1086.503,135.628,432.684,175.210,20.590,153.304
C09669=1086.509,135.878,432.664,175.212,20.592,153.304
C09670=1086.515,136.127,432.644,175.214,20.594,153.304
C09671=1086.520,136.376,432.623,175.217,20.595,153.304
C09672=1086.526,136.625,432.603,175.219,20.597,153.304
C09673=1086.532,136.874,432.584,175.221,20.598,153.304
C09674=1086.537,137.123,432.564,175.223,20.600,153.304
C09675=1086.543,137.372,432.544,175.226,20.602,153.304
C09676=1086.548,137.621,432.523,175.228,20.603,153.304
C09677=1086.554,137.871,432.504,175.230,20.605,153.304
C09678=1086.559,138.120,432.483,175.232,20.606,153.304
C09679=1086.565,138.369,432.463,175.235,20.608,153.304
C09680=1086.571,138.618,432.443,175.237,20.610,153.304
C09681=1086.577,138.867,432.423,175.239,20.611,153.304
C09682=1086.582,139.116,432.402,175.241,20.613,153.304
C09683=1086.588,139.365,432.383,175.244,20.614,153.304
C09684=1086.593,139.614,432.363,175.245,20.616,153.304
C09685=1086.599,139.864,432.342,175.247,20.618,153.304
C09686=1086.605,140.113,432.322,175.250,20.619,153.304
C09687=1086.611,140.362,432.302,175.252,20.621,153.304
C09688=1086.616,140.611,432.281,175.254,20.622,153.304
C09689=1086.621,140.860,432.261,175.257,20.624,153.304
C09690=1086.627,141.109,432.241,175.259,20.626,153.304
C09691=1086.632,141.358,432.220,175.261,20.627,153.303
C09692=1086.638,141.607,432.200,175.264,20.629,153.303
C09693=1086.644,141.856,432.180,175.266,20.630,153.303
C09694=1086.649,142.105,432.159,175.268,20.632,153.303
C09695=1086.655,142.354,432.139,175.270,20.634,153.303
C09696=1086.661,142.604,432.118,175.273,20.636,153.303
C09697=1086.666,142.853,432.098,175.274,20.637,153.303
C09698=1086.672,143.102,432.078,175.277,20.639,153.303
C09699=1086.678,143.380,432.055,175.279,20.640,153.303
C09700=1086.684,143.658,432.032,175.282,20.642,153.303
C09701=1086.690,143.938,432.009,175.284,20.644,153.303
C09702=1086.696,144.216,431.986,175.287,20.646,153.303
C09703=1086.702,144.465,431.966,175.289,20.647,153.303
C09704=1086.708,144.713,431.946,175.292,20.649,153.303
C09705=1086.713,144.963,431.925,175.294,20.651,153.303
C09706=1086.719,145.212,431.904,175.297,20.653,153.303
C09707=1086.725,145.461,431.884,175.298,20.653,153.303
C09708=1086.730,145.710,431.864,175.301,20.655,153.303
C09709=1086.735,145.959,431.843,175.303,20.657,153.303
C09710=1086.741,146.208,431.823,175.306,20.659,153.303
C09711=1086.748,146.457,431.802,175.307,20.660,153.303
C09712=1086.753,146.707,431.781,175.310,20.662,153.303
C09713=1086.758,146.956,431.760,175.312,20.663,153.302
C09714=1086.764,147.205,431.740,175.315,20.665,153.303
C09715=1086.769,147.454,431.720,175.317,20.666,153.302
C09716=1086.775,147.703,431.699,175.319,20.668,153.302
C09717=1086.781,147.952,431.678,175.321,20.669,153.302
C09718=1086.787,148.201,431.658,175.324,20.671,153.302
C09719=1086.792,148.450,431.637,175.326,20.673,153.302
C09720=1086.797,148.699,431.617,175.329,20.674,153.302
C09721=1086.803,148.949,431.596,175.330,20.676,153.302
C09722=1086.809,149.197,431.574,175.333,20.677,153.302
C09723=1086.815,149.446,431.555,175.335,20.679,153.302
C09724=1086.820,149.695,431.534,175.338,20.680,153.302
C09725=1086.826,149.945,431.512,175.340,20.682,153.302
C09726=1086.831,150.194,431.492,175.342,20.683,153.302
C09727=1086.837,150.443,431.471,175.344,20.685,153.302
C09728=1086.842,150.692,431.451,175.347,20.687,153.302
C09729=1086.848,150.941,431.429,175.349,20.689,153.302
C09730=1086.853,151.190,431.408,175.352,20.690,153.302
C09731=1086.859,151.439,431.389,175.354,20.691,153.302
C09732=1086.865,151.688,431.367,175.356,20.693,153.302
C09733=1086.871,151.937,431.346,175.359,20.694,153.301
C09734=1086.876,152.186,431.326,175.361,20.696,153.301
C09735=1086.881,152.435,431.305,175.364,20.698,153.301
C09736=1086.887,152.684,431.284,175.365,20.699,153.301
C09737=1086.893,152.933,431.262,175.368,20.701,153.301
C09738=1086.898,153.182,431.242,175.370,20.702,153.301
C09739=1086.903,153.432,431.221,175.373,20.704,153.301
C09740=1086.910,153.681,431.200,175.375,20.705,153.301
C09741=1086.915,153.930,431.179,175.378,20.707,153.301
C09742=1086.920,154.178,431.158,175.379,20.708,153.301
C09743=1086.926,154.428,431.137,175.382,20.710,153.301
C09744=1086.932,154.677,431.116,175.384,20.712,153.301
C09745=1086.937,154.926,431.095,175.387,20.713,153.301
C09746=1086.943,155.174,431.074,175.390,20.715,153.301
C09747=1086.948,155.424,431.053,175.392,20.717,153.301
C09748=1086.954,155.673,431.032,175.394,20.717,153.301
C09749=1086.959,155.922,431.011,175.396,20.719,153.301
C09750=1086.965,156.171,430.989,175.399,20.721,153.300
C09751=1086.971,156.420,430.969,175.401,20.722,153.300
C09752=1086.976,156.669,430.948,175.404,20.724,153.300
C09753=1086.982,156.918,430.927,175.406,20.726,153.300
C09754=1086.988,157.167,430.905,175.408,20.727,153.300
C09755=1086.993,157.416,430.885,175.410,20.729,153.300
C09756=1086.999,157.665,430.863,175.413,20.730,153.300
C09757=1087.004,157.914,430.841,175.415,20.732,153.300
C09758=1087.010,158.164,430.820,175.418,20.733,153.300
C09759=1087.015,158.412,430.799,175.420,20.735,153.300
C09760=1087.021,158.662,430.779,175.423,20.737,153.300
C09761=1087.027,158.911,430.757,175.424,20.738,153.300
C09762=1087.032,159.159,430.736,175.427,20.739,153.300
C09763=1087.038,159.437,430.713,175.430,20.741,153.299
C09764=1087.044,159.716,430.688,175.433,20.743,153.299
C09765=1087.051,159.994,430.665,175.436,20.744,153.299
C09766=1087.058,160.272,430.641,175.438,20.746,153.299
C09767=1087.062,160.521,430.619,175.440,20.748,153.299
C09768=1087.068,160.771,430.598,175.443,20.749,153.299
C09769=1087.074,161.019,430.577,175.446,20.751,153.299
C09770=1087.080,161.269,430.555,175.448,20.753,153.299
C09771=1087.086,161.517,430.534,175.450,20.753,153.299
C09772=1087.090,161.767,430.513,175.452,20.755,153.299
C09773=1087.096,162.016,430.491,175.455,20.757,153.299
C09774=1087.102,162.264,430.470,175.457,20.758,153.299
C09775=1087.107,162.513,430.448,175.460,20.760,153.299
C09776=1087.113,162.762,430.427,175.462,20.762,153.299
C09777=1087.117,163.012,430.405,175.465,20.763,153.298
C09778=1087.123,163.261,430.384,175.467,20.765,153.298
C09779=1087.129,163.509,430.363,175.469,20.766,153.298
C09780=1087.134,163.758,430.341,175.472,20.767,153.298
C09781=1087.140,164.007,430.319,175.474,20.769,153.298
C09782=1087.144,164.257,430.298,175.477,20.771,153.298
C09783=1087.151,164.506,430.276,175.479,20.773,153.298
C09784=1087.156,164.755,430.255,175.481,20.774,153.298
C09785=1087.161,165.003,430.233,175.484,20.776,153.298
C09786=1087.167,165.253,430.212,175.486,20.777,153.298
C09787=1087.172,165.501,430.190,175.489,20.779,153.298
C09788=1087.178,165.751,430.168,175.491,20.780,153.298
C09789=1087.183,165.999,430.146,175.493,20.782,153.298
C09790=1087.189,166.248,430.125,175.496,20.783,153.298
C09791=1087.194,166.498,430.103,175.498,20.785,153.298
C09792=1087.199,166.747,430.082,175.501,20.787,153.298
C09793=1087.205,166.996,430.060,175.503,20.788,153.297
C09794=1087.210,167.245,430.039,175.506,20.789,153.297
C09795=1087.216,167.494,430.016,175.508,20.791,153.297
C09796=1087.221,167.743,429.995,175.511,20.793,153.297
C09797=1087.227,167.992,429.973,175.513,20.794,153.297
C09798=1087.232,168.241,429.952,175.516,20.796,153.297
C09799=1087.238,168.490,429.929,175.518,20.797,153.297
C09800=1087.243,168.739,429.908,175.520,20.799,153.297
C09801=1087.249,168.988,429.885,175.523,20.800,153.297
C09802=1087.255,169.236,429.864,175.525,20.801,153.297
C09803=1087.260,169.486,429.842,175.528,20.803,153.297
C09804=1087.265,169.734,429.820,175.530,20.805,153.297
C09805=1087.271,169.984,429.798,175.533,20.806,153.296
C09806=1087.276,170.232,429.777,175.535,20.808,153.296
C09807=1087.282,170.482,429.755,175.538,20.809,153.296
C09808=1087.287,170.730,429.733,175.540,20.811,153.296
C09809=1087.293,170.980,429.711,175.543,20.812,153.296
C09810=1087.299,171.229,429.690,175.546,20.814,153.296
C09811=1087.304,171.477,429.667,175.548,20.815,153.296
C09812=1087.310,171.726,429.645,175.550,20.817,153.296
C09813=1087.315,171.975,429.623,175.552,20.818,153.296
C09814=1087.321,172.224,429.602,175.555,20.820,153.296
C09815=1087.326,172.473,429.580,175.557,20.821,153.296
C09816=1087.332,172.722,429.557,175.560,20.823,153.295
C09817=1087.338,172.971,429.535,175.563,20.824,153.295
C09818=1087.343,173.220,429.513,175.565,20.826,153.295
C09819=1087.349,173.469,429.492,175.568,20.827,153.295
C09820=1087.354,173.718,429.470,175.570,20.829,153.295
C09821=1087.360,173.967,429.448,175.573,20.830,153.295
C09822=1087.366,174.216,429.425,175.575,20.832,153.295
C09823=1087.371,174.465,429.404,175.578,20.833,153.295
C09824=1087.377,174.714,429.381,175.581,20.834,153.295
C09825=1087.382,174.963,429.359,175.583,20.836,153.295
C09826=1087.388,175.212,429.338,175.586,20.838,153.295
C09827=1087.394,175.490,429.313,175.588,20.839,153.294
C09828=1087.400,175.767,429.288,175.591,20.841,153.294
C09829=1087.407,176.045,429.263,175.594,20.843,153.294
C09830=1087.413,176.324,429.238,175.597,20.844,153.294
C09831=1087.419,176.572,429.216,175.599,20.845,153.294
C09832=1087.424,176.821,429.194,175.602,20.847,153.294
C09833=1087.430,177.071,429.172,175.605,20.848,153.294
C09834=1087.435,177.319,429.150,175.607,20.850,153.294
C09835=1087.441,177.568,429.127,175.610,20.851,153.293
C09836=1087.447,177.817,429.105,175.612,20.853,153.293
C09837=1087.452,178.065,429.083,175.615,20.855,153.293
C09838=1087.458,178.315,429.061,175.617,20.856,153.293
C09839=1087.464,178.564,429.039,175.620,20.857,153.293
C09840=1087.470,178.813,429.016,175.622,20.859,153.293
C09841=1087.475,179.061,428.994,175.625,20.860,153.293
C09842=1087.481,179.311,428.972,175.628,20.862,153.293
C09843=1087.487,179.559,428.949,175.630,20.863,153.293
C09844=1087.492,179.809,428.927,175.633,20.865,153.293
C09845=1087.497,180.057,428.904,175.635,20.866,153.292
C09846=1087.503,180.306,428.883,175.637,20.867,153.292
C09847=1087.509,180.555,428.860,175.640,20.868,153.292
C09848=1087.514,180.805,428.838,175.642,20.870,153.292
C09849=1087.521,181.053,428.815,175.645,20.871,153.292
C09850=1087.526,181.302,428.793,175.648,20.873,153.292
C09851=1087.531,181.551,428.771,175.650,20.874,153.292
C09852=1087.538,181.800,428.748,175.653,20.876,153.292
C09853=1087.543,182.049,428.726,175.655,20.877,153.292
C09854=1087.549,182.298,428.703,175.658,20.878,153.291
C09855=1087.554,182.546,428.680,175.661,20.879,153.291
C09856=1087.560,182.795,428.659,175.663,20.881,153.291
C09857=1087.566,183.044,428.636,175.666,20.882,153.291
C09858=1087.572,183.293,428.613,175.668,20.884,153.291
C09859=1087.577,183.543,428.591,175.671,20.885,153.291
C09860=1087.584,183.791,428.568,175.674,20.887,153.291
C09861=1087.589,184.040,428.545,175.677,20.888,153.290
C09862=1087.594,184.289,428.523,175.680,20.890,153.290
C09863=1087.600,184.538,428.501,175.682,20.891,153.290
C09864=1087.606,184.787,428.478,175.685,20.893,153.290
C09865=1087.612,185.035,428.455,175.688,20.894,153.290
C09866=1087.618,185.285,428.433,175.690,20.896,153.290
C09867=1087.623,185.534,428.410,175.693,20.897,153.290
C09868=1087.628,185.782,428.387,175.695,20.898,153.290
C09869=1087.633,186.031,428.364,175.698,20.900,153.289
C09870=1087.639,186.281,428.342,175.700,20.901,153.289
C09871=1087.645,186.530,428.319,175.703,20.903,153.289
C09872=1087.650,186.778,428.296,175.705,20.905,153.289
C09873=1087.655,187.027,428.273,175.708,20.906,153.289
C09874=1087.661,187.276,428.250,175.711,20.908,153.289
C09875=1087.667,187.525,428.228,175.713,20.909,153.289
C09876=1087.672,187.774,428.205,175.716,20.910,153.289
C09877=1087.678,188.022,428.183,175.718,20.912,153.289
C09878=1087.682,188.271,428.159,175.721,20.913,153.289
C09879=1087.688,188.520,428.136,175.724,20.915,153.288
C09880=1087.694,188.769,428.113,175.726,20.916,153.288
C09881=1087.700,189.018,428.090,175.729,20.918,153.288
C09882=1087.705,189.267,428.067,175.731,20.919,153.288
C09883=1087.711,189.515,428.045,175.734,20.920,153.288
C09884=1087.715,189.765,428.022,175.736,20.922,153.288
C09885=1087.721,190.014,427.999,175.739,20.924,153.288
C09886=1087.727,190.263,427.976,175.742,20.925,153.288
C09887=1087.732,190.512,427.953,175.745,20.927,153.288
C09888=1087.738,190.761,427.930,175.748,20.929,153.288
C09889=1087.744,191.010,427.907,175.750,20.930,153.287
C09890=1087.748,191.258,427.884,175.753,20.931,153.287
C09891=1087.755,191.536,427.858,175.755,20.933,153.287
C09892=1087.762,191.813,427.832,175.759,20.935,153.287
C09893=1087.767,192.090,427.806,175.761,20.936,153.287
C09894=1087.774,192.368,427.781,175.764,20.938,153.287
C09895=1087.779,192.617,427.758,175.767,20.940,153.287
C09896=1087.785,192.866,427.735,175.770,20.941,153.287
C09897=1087.790,193.115,427.711,175.773,20.942,153.286
C09898=1087.796,193.364,427.689,175.775,20.944,153.286
C09899=1087.802,193.613,427.666,175.778,20.945,153.286
C09900=1087.808,193.861,427.642,175.780,20.947,153.286
C09901=1087.813,194.110,427.618,175.783,20.948,153.286
C09902=1087.818,194.359,427.595,175.786,20.950,153.286
C09903=1087.824,194.608,427.572,175.788,20.951,153.286
C09904=1087.829,194.856,427.550,175.791,20.952,153.286
C09905=1087.834,195.106,427.526,175.794,20.953,153.285
C09906=1087.840,195.354,427.503,175.796,20.955,153.285
C09907=1087.846,195.603,427.480,175.800,20.957,153.285
C09908=1087.852,195.852,427.457,175.802,20.958,153.285
C09909=1087.857,196.101,427.433,175.805,20.960,153.285
C09910=1087.862,196.350,427.410,175.807,20.961,153.285
C09911=1087.869,196.599,427.386,175.810,20.962,153.285
C09912=1087.874,196.848,427.363,175.813,20.964,153.285
C09913=1087.880,197.097,427.340,175.815,20.965,153.284
C09914=1087.885,197.346,427.317,175.818,20.967,153.284
C09915=1087.892,197.594,427.293,175.820,20.968,153.284
C09916=1087.897,197.843,427.270,175.824,20.970,153.284
C09917=1087.902,198.092,427.247,175.827,20.971,153.284
C09918=1087.908,198.340,427.223,175.829,20.972,153.284
C09919=1087.913,198.590,427.200,175.832,20.974,153.284
C09920=1087.919,198.838,427.177,175.834,20.975,153.284
C09921=1087.925,199.087,427.153,175.837,20.977,153.283
C09922=1087.930,199.336,427.129,175.840,20.978,153.283
C09923=1087.936,199.585,427.106,175.842,20.980,153.283
C09924=1087.942,199.833,427.083,175.846,20.982,153.283
C09925=1087.947,200.082,427.059,175.849,20.982,153.283
C09926=1087.953,200.331,427.035,175.851,20.984,153.283
C09927=1087.959,200.580,427.012,175.854,20.985,153.283
C09928=1087.964,200.829,426.989,175.856,20.987,153.282
C09929=1087.970,201.078,426.965,175.859,20.988,153.282
C09930=1087.975,201.327,426.942,175.861,20.990,153.282
C09931=1087.981,201.575,426.918,175.864,20.991,153.282
C09932=1087.987,201.824,426.895,175.868,20.992,153.282
C09933=1087.993,202.073,426.870,175.870,20.994,153.282
C09934=1087.999,202.322,426.847,175.873,20.995,153.282
C09935=1088.005,202.570,426.824,175.876,20.997,153.281
C09936=1088.010,202.820,426.800,175.878,20.998,153.281
C09937=1088.016,203.068,426.776,175.881,21.000,153.281
C09938=1088.021,203.317,426.753,175.883,21.001,153.281
C09939=1088.026,203.566,426.729,175.887,21.003,153.281
C09940=1088.032,203.814,426.705,175.889,21.004,153.281
C09941=1088.038,204.064,426.681,175.892,21.005,153.281
C09942=1088.044,204.312,426.657,175.895,21.007,153.281
C09943=1088.049,204.561,426.634,175.897,21.008,153.280
C09944=1088.054,204.810,426.610,175.900,21.010,153.280
C09945=1088.060,205.058,426.586,175.903,21.012,153.280
C09946=1088.065,205.308,426.562,175.906,21.013,153.280
C09947=1088.071,205.556,426.539,175.909,21.014,153.280
C09948=1088.077,205.805,426.514,175.911,21.016,153.280
C09949=1088.082,206.054,426.491,175.914,21.017,153.280
C09950=1088.088,206.303,426.467,175.917,21.019,153.280
C09951=1088.093,206.551,426.443,175.920,21.021,153.279
C09952=1088.098,206.800,426.419,175.922,21.022,153.279
C09953=1088.104,207.049,426.395,175.925,21.023,153.279
C09954=1088.110,207.298,426.371,175.928,21.024,153.279
C09955=1088.133,208.322,426.272,176.002,21.062,153.275
C09956=1088.140,208.636,426.242,176.005,21.065,153.275
C09957=1088.148,208.950,426.211,176.008,21.068,153.276
C09958=1088.154,209.265,426.180,176.012,21.071,153.276
C09959=1088.161,209.579,426.150,176.016,21.074,153.276
C09960=1088.167,209.828,426.125,176.018,21.077,153.276
C09961=1088.172,210.076,426.101,176.021,21.079,153.276
C09962=1088.178,210.325,426.076,176.023,21.081,153.276
C09963=1088.184,210.574,426.052,176.026,21.084,153.276
C09964=1088.190,210.822,426.027,176.029,21.086,153.276
C09965=1088.196,211.071,426.003,176.031,21.088,153.276
C09966=1088.201,211.320,425.979,176.034,21.091,153.276
C09967=1088.206,211.568,425.954,176.036,21.093,153.276
C09968=1088.212,211.818,425.930,176.039,21.096,153.276
C09969=1088.218,212.066,425.905,176.042,21.098,153.276
C09970=1088.224,212.315,425.880,176.045,21.101,153.277
C09971=1088.229,212.564,425.856,176.047,21.103,153.277
C09972=1088.234,212.812,425.832,176.050,21.105,153.277
C09973=1088.240,213.061,425.807,176.053,21.107,153.277
C09974=1088.246,213.309,425.782,176.056,21.110,153.277
C09975=1088.252,213.559,425.757,176.058,21.112,153.277
C09976=1088.256,213.808,425.732,176.060,21.115,153.277
C09977=1088.263,214.056,425.707,176.064,21.117,153.277
C09978=1088.268,214.305,425.683,176.066,21.119,153.277
C09979=1088.273,214.553,425.659,176.069,21.122,153.277
C09980=1088.279,214.802,425.633,176.071,21.124,153.278
C09981=1088.285,215.051,425.609,176.074,21.127,153.278
C09982=1088.291,215.300,425.584,176.077,21.129,153.278
C09983=1088.296,215.548,425.559,176.080,21.131,153.278
C09984=1088.303,215.867,425.527,176.083,21.134,153.278
C09985=1088.310,216.185,425.496,176.087,21.138,153.278
C09986=1088.317,216.504,425.464,176.090,21.141,153.278
C09987=1088.324,216.822,425.433,176.094,21.144,153.278
C09988=1088.330,217.071,425.407,176.096,21.146,153.278
C09989=1088.336,217.319,425.383,176.098,21.148,153.278
C09990=1088.341,217.568,425.357,176.101,21.151,153.279
C09991=1088.346,217.817,425.333,176.104,21.153,153.279
C09992=1088.353,218.065,425.307,176.107,21.156,153.279
C09993=1088.359,218.315,425.283,176.109,21.158,153.279
C09994=1088.364,218.563,425.258,176.112,21.161,153.279
C09995=1088.369,218.812,425.233,176.115,21.163,153.279
C09996=1088.375,219.060,425.208,176.118,21.166,153.279
//INST
///DATE 2021/06/25 14:44
///ATTR SC,RW,RJ
////FRAME ROBOT
///GROUP1 RB1
NOP
MOVL C00000 V=800.0 PL=0
MOVL C00001 V=800.0 PL=0
MOVL C00002 V=800.0 PL=0
MOVL C00003 V=800.0 PL=0
MOVL C00004 V=800.0 PL=0
MOVL C00005 V=800.0 PL=0
MOVL C00006 V=800.0 PL=0
MOVL C00007 V=800.0 PL=0
MOVL C00008 V=800.0 PL=0
MOVL C00009 V=800.0 PL=0
MOVL C00010 V=800.0 PL=0
MOVL C00011 V=800.0 PL=0
MOVL C00012 V=800.0 PL=0
MOVL C00013 V=800.0 PL=0
MOVL C00014 V=800.0 PL=0
MOVL C00015 V=800.0 PL=0
MOVL C00016 V=800.0 PL=0
MOVL C00017 V=800.0 PL=0
MOVL C00018 V=800.0 PL=0
MOVL C00019 V=800.0 PL=0
MOVL C00020 V=800.0 PL=0
MOVL C00021 V=800.0 PL=0
MOVL C00022 V=800.0 PL=0
MOVL C00023 V=800.0 PL=0
MOVL C00024 V=800.0 PL=0
MOVL C00025 V=800.0 PL=0
MOVL C00026 V=800.0 PL=0
MOVL C00027 V=800.0 PL=0
MOVL C00028 V=800.0 PL=0
MOVL C00029 V=800.0 PL=0
MOVL C00030 V=800.0 PL=0
MOVL C00031 V=800.0 PL=0
MOVL C00032 V=800.0 PL=0
MOVL C00033 V=800.0 PL=0
MOVL C00034 V=800.0 PL=0
MOVL C00035 V=800.0 PL=0
MOVL C00036 V=800.0 PL=0
MOVL C00037 V=800.0 PL=0
MOVL C00038 V=800.0 PL=0
MOVL C00039 V=800.0 PL=0
MOVL C00040 V=800.0 PL=0
MOVL C00041 V=800.0 PL=0
MOVL C00042 V=800.0 PL=0
MOVL C00043 V=800.0 PL=0
MOVL C00044 V=800.0 PL=0
MOVL C00045 V=800.0 PL=0
MOVL C00046 V=800.0 PL=0
MOVL C00047 V=800.0 PL=0
MOVL C00048 V=800.0 PL=0
MOVL C00049 V=800.0 PL=0
MOVL C00050 V=800.0 PL=0
MOVL C00051 V=800.0 PL=0
MOVL C00052 V=800.0 PL=0
MOVL C00053 V=800.0 PL=0
MOVL C00054 V=800.0 PL=0
MOVL C00055 V=800.0 PL=0
MOVL C00056 V=800.0 PL=0
MOVL C00057 V=800.0 PL=0
MOVL C00058 V=800.0 PL=0
MOVL C00059 V=800.0 PL=0
MOVL C00060 V=800.0 PL=0
MOVL C00061 V=800.0 PL=0
MOVL C00062 V=800.0 PL=0
MOVL C00063 V=800.0 PL=0
MOVL C00064 V=800.0 PL=0
MOVL C00065 V=800.0 PL=0
MOVL C00066 V=800.0 PL=0
MOVL C00067 V=800.0 PL=0
MOVL C00068 V=800.0 PL=0
MOVL C00069 V=800.0 PL=0
MOVL C00070 V=800.0 PL=0
MOVL C00071 V=800.0 PL=0
MOVL C00072 V=800.0 PL=0
MOVL C00073 V=800.0 PL=0
MOVL C00074 V=800.0 PL=0
MOVL C00075 V=800.0 PL=0
MOVL C00076 V=800.0 PL=0
MOVL C00077 V=800.0 PL=0
MOVL C00078 V=800.0 PL=0
MOVL C00079 V=800.0 PL=0
MOVL C00080 V=800.0 PL=0
MOVL C00081 V=800.0 PL=0
MOVL C00082 V=800.0 PL=0
MOVL C00083 V=800.0 PL=0
MOVL C00084 V=800.0 PL=0
MOVL C00085 V=800.0 PL=0
MOVL C00086 V=800.0 PL=0
MOVL C00087 V=800.0 PL=0
MOVL C00088 V=800.0 PL=0
MOVL C00089 V=800.0 PL=0
MOVL C00090 V=800.0 PL=0
MOVL C00091 V=800.0 PL=0
MOVL C00092 V=800.0 PL=0
MOVL C00093 V=800.0 PL=0
MOVL C00094 V=800.0 PL=0
MOVL C00095 V=800.0 PL=0
MOVL C00096 V=800.0 PL=0
MOVL C00097 V=800.0 PL=0
MOVL C00098 V=800.0 PL=0
MOVL C00099 V=800.0 PL=0
MOVL C00100 V=800.0 PL=0
MOVL C00101 V=800.0 PL=0
MOVL C00102 V=800.0 PL=0
MOVL C00103 V=800.0 PL=0
MOVL C00104 V=800.0 PL=0
MOVL C00105 V=800.0 PL=0
MOVL C00106 V=800.0 PL=0
MOVL C00107 V=800.0 PL=0
MOVL C00108 V=800.0 PL=0
MOVL C00109 V=800.0 PL=0
MOVL C00110 V=800.0 PL=0
MOVL C00111 V=800.0 PL=0
MOVL C00112 V=800.0 PL=0
MOVL C00113 V=800.0 PL=0
MOVL C00114 V=800.0 PL=0
MOVL C00115 V=800.0 PL=0
MOVL C00116 V=800.0 PL=0
MOVL C00117 V=800.0 PL=0
MOVL C00118 V=800.0 PL=0
MOVL C00119 V=800.0 PL=0
MOVL C00120 V=800.0 PL=0
MOVL C00121 V=800.0 PL=0
MOVL C00122 V=800.0 PL=0
MOVL C00123 V=800.0 PL=0
MOVL C00124 V=800.0 PL=0
MOVL C00125 V=800.0 PL=0
MOVL C00126 V=800.0 PL=0
MOVL C00127 V=800.0 PL=0
MOVL C00128 V=800.0 PL=0
MOVL C00129 V=800.0 PL=0
MOVL C00130 V=800.0 PL=0
MOVL C00131 V=800.0 PL=0
MOVL C00132 V=800.0 PL=0
MOVL C00133 V=800.0 PL=0
MOVL C00134 V=800.0 PL=0
MOVL C00135 V=800.0 PL=0
MOVL C00136 V=800.0 PL=0
MOVL C00137 V=800.0 PL=0
MOVL C00138 V=800.0 PL=0
MOVL C00139 V=800.0 PL=0
MOVL C00140 V=800.0 PL=0
MOVL C00141 V=800.0 PL=0
MOVL C00142 V=800.0 PL=0
MOVL C00143 V=800.0 PL=0
MOVL C00144 V=800.0 PL=0
MOVL C00145 V=800.0 PL=0
MOVL C00146 V=800.0 PL=0
MOVL C00147 V=800.0 PL=0
MOVL C00148 V=800.0 PL=0
MOVL C00149 V=800.0 PL=0
MOVL C00150 V=800.0 PL=0
MOVL C00151 V=800.0 PL=0
MOVL C00152 V=800.0 PL=0
MOVL C00153 V=800.0 PL=0
MOVL C00154 V=800.0 PL=0
MOVL C00155 V=800.0 PL=0
MOVL C00156 V=800.0 PL=0
MOVL C00157 V=800.0 PL=0
MOVL C00158 V=800.0 PL=0
MOVL C00159 V=800.0 PL=0
MOVL C00160 V=800.0 PL=0
MOVL C00161 V=800.0 PL=0
MOVL C00162 V=800.0 PL=0
MOVL C00163 V=800.0 PL=0
MOVL C00164 V=800.0 PL=0
MOVL C00165 V=800.0 PL=0
MOVL C00166 V=800.0 PL=0
MOVL C00167 V=800.0 PL=0
MOVL C00168 V=800.0 PL=0
MOVL C00169 V=800.0 PL=0
MOVL C00170 V=800.0 PL=0
MOVL C00171 V=800.0 PL=0
MOVL C00172 V=800.0 PL=0
MOVL C00173 V=800.0 PL=0
MOVL C00174 V=800.0 PL=0
MOVL C00175 V=800.0 PL=0
MOVL C00176 V=800.0 PL=0
MOVL C00177 V=800.0 PL=0
MOVL C00178 V=800.0 PL=0
MOVL C00179 V=800.0 PL=0
MOVL C00180 V=800.0 PL=0
MOVL C00181 V=800.0 PL=0
MOVL C00182 V=800.0 PL=0
MOVL C00183 V=800.0 PL=0
MOVL C00184 V=800.0 PL=0
MOVL C00185 V=800.0 PL=0
MOVL C00186 V=800.0 PL=0
MOVL C00187 V=800.0 PL=0
MOVL C00188 V=800.0 PL=0
MOVL C00189 V=800.0 PL=0
MOVL C00190 V=800.0 PL=0
MOVL C00191 V=800.0 PL=0
MOVL C00192 V=800.0 PL=0
MOVL C00193 V=800.0 PL=0
MOVL C00194 V=800.0 PL=0
MOVL C00195 V=800.0 PL=0
MOVL C00196 V=800.0 PL=0
MOVL C00197 V=800.0 PL=0
MOVL C00198 V=800.0 PL=0
MOVL C00199 V=800.0 PL=0
MOVL C00200 V=800.0 PL=0
MOVL C00201 V=800.0 PL=0
MOVL C00202 V=800.0 PL=0
MOVL C00203 V=800.0 PL=0
MOVL C00204 V=800.0 PL=0
MOVL C00205 V=800.0 PL=0
MOVL C00206 V=800.0 PL=0
MOVL C00207 V=800.0 PL=0
MOVL C00208 V=800.0 PL=0
MOVL C00209 V=800.0 PL=0
MOVL C00210 V=800.0 PL=0
MOVL C00211 V=800.0 PL=0
MOVL C00212 V=800.0 PL=0
MOVL C00213 V=800.0 PL=0
MOVL C00214 V=800.0 PL=0
MOVL C00215 V=800.0 PL=0
MOVL C00216 V=800.0 PL=0
MOVL C00217 V=800.0 PL=0
MOVL C00218 V=800.0 PL=0
MOVL C00219 V=800.0 PL=0
MOVL C00220 V=800.0 PL=0
MOVL C00221 V=800.0 PL=0
MOVL C00222 V=800.0 PL=0
MOVL C00223 V=800.0 PL=0
MOVL C00224 V=800.0 PL=0
MOVL C00225 V=800.0 PL=0
MOVL C00226 V=800.0 PL=0
MOVL C00227 V=800.0 PL=0
MOVL C00228 V=800.0 PL=0
MOVL C00229 V=800.0 PL=0
MOVL C00230 V=800.0 PL=0
MOVL C00231 V=800.0 PL=0
MOVL C00232 V=800.0 PL=0
MOVL C00233 V=800.0 PL=0
MOVL C00234 V=800.0 PL=0
MOVL C00235 V=800.0 PL=0
MOVL C00236 V=800.0 PL=0
MOVL C00237 V=800.0 PL=0
MOVL C00238 V=800.0 PL=0
MOVL C00239 V=800.0 PL=0
MOVL C00240 V=800.0 PL=0
MOVL C00241 V=800.0 PL=0
MOVL C00242 V=800.0 PL=0
MOVL C00243 V=800.0 PL=0
MOVL C00244 V=800.0 PL=0
MOVL C00245 V=800.0 PL=0
MOVL C00246 V=800.0 PL=0
MOVL C00247 V=800.0 PL=0
MOVL C00248 V=800.0 PL=0
MOVL C00249 V=800.0 PL=0
MOVL C00250 V=800.0 PL=0
MOVL C00251 V=800.0 PL=0
MOVL C00252 V=800.0 PL=0
MOVL C00253 V=800.0 PL=0
MOVL C00254 V=800.0 PL=0
MOVL C00255 V=800.0 PL=0
MOVL C00256 V=800.0 PL=0
MOVL C00257 V=800.0 PL=0
MOVL C00258 V=800.0 PL=0
MOVL C00259 V=800.0 PL=0
MOVL C00260 V=800.0 PL=0
MOVL C00261 V=800.0 PL=0
MOVL C00262 V=800.0 PL=0
MOVL C00263 V=800.0 PL=0
MOVL C00264 V=800.0 PL=0
MOVL C00265 V=800.0 PL=0
MOVL C00266 V=800.0 PL=0
MOVL C00267 V=800.0 PL=0
MOVL C00268 V=800.0 PL=0
MOVL C00269 V=800.0 PL=0
MOVL C00270 V=800.0 PL=0
MOVL C00271 V=800.0 PL=0
MOVL C00272 V=800.0 PL=0
MOVL C00273 V=800.0 PL=0
MOVL C00274 V=800.0 PL=0
MOVL C00275 V=800.0 PL=0
MOVL C00276 V=800.0 PL=0
MOVL C00277 V=800.0 PL=0
MOVL C00278 V=800.0 PL=0
MOVL C00279 V=800.0 PL=0
MOVL C00280 V=800.0 PL=0
MOVL C00281 V=800.0 PL=0
MOVL C00282 V=800.0 PL=0
MOVL C00283 V=800.0 PL=0
MOVL C00284 V=800.0 PL=0
MOVL C00285 V=800.0 PL=0
MOVL C00286 V=800.0 PL=0
MOVL C00287 V=800.0 PL=0
MOVL C00288 V=800.0 PL=0
MOVL C00289 V=800.0 PL=0
MOVL C00290 V=800.0 PL=0
MOVL C00291 V=800.0 PL=0
MOVL C00292 V=800.0 PL=0
MOVL C00293 V=800.0 PL=0
MOVL C00294 V=800.0 PL=0
MOVL C00295 V=800.0 PL=0
MOVL C00296 V=800.0 PL=0
MOVL C00297 V=800.0 PL=0
MOVL C00298 V=800.0 PL=0
MOVL C00299 V=800.0 PL=0
MOVL C00300 V=800.0 PL=0
MOVL C00301 V=800.0 PL=0
MOVL C00302 V=800.0 PL=0
MOVL C00303 V=800.0 PL=0
MOVL C00304 V=800.0 PL=0
MOVL C00305 V=800.0 PL=0
MOVL C00306 V=800.0 PL=0
MOVL C00307 V=800.0 PL=0
MOVL C00308 V=800.0 PL=0
MOVL C00309 V=800.0 PL=0
MOVL C00310 V=800.0 PL=0
MOVL C00311 V=800.0 PL=0
MOVL C00312 V=800.0 PL=0
MOVL C00313 V=800.0 PL=0
MOVL C00314 V=800.0 PL=0
MOVL C00315 V=800.0 PL=0
MOVL C00316 V=800.0 PL=0
MOVL C00317 V=800.0 PL=0
MOVL C00318 V=800.0 PL=0
MOVL C00319 V=800.0 PL=0
MOVL C00320 V=800.0 PL=0
MOVL C00321 V=800.0 PL=0
MOVL C00322 V=800.0 PL=0
MOVL C00323 V=800.0 PL=0
MOVL C00324 V=800.0 PL=0
MOVL C00325 V=800.0 PL=0
MOVL C00326 V=800.0 PL=0
MOVL C00327 V=800.0 PL=0
MOVL C00328 V=800.0 PL=0
MOVL C00329 V=800.0 PL=0
MOVL C00330 V=800.0 PL=0
MOVL C00331 V=800.0 PL=0
MOVL C00332 V=800.0 PL=0
MOVL C00333 V=800.0 PL=0
MOVL C00334 V=800.0 PL=0
MOVL C00335 V=800.0 PL=0
MOVL C00336 V=800.0 PL=0
MOVL C00337 V=800.0 PL=0
MOVL C00338 V=800.0 PL=0
MOVL C00339 V=800.0 PL=0
MOVL C00340 V=800.0 PL=0
MOVL C00341 V=800.0 PL=0
MOVL C00342 V=800.0 PL=0
MOVL C00343 V=800.0 PL=0
MOVL C00344 V=800.0 PL=0
MOVL C00345 V=800.0 PL=0
MOVL C00346 V=800.0 PL=0
MOVL C00347 V=800.0 PL=0
MOVL C00348 V=800.0 PL=0
MOVL C00349 V=800.0 PL=0
MOVL C00350 V=800.0 PL=0
MOVL C00351 V=800.0 PL=0
MOVL C00352 V=800.0 PL=0
MOVL C00353 V=800.0 PL=0
MOVL C00354 V=800.0 PL=0
MOVL C00355 V=800.0 PL=0
MOVL C00356 V=800.0 PL=0
MOVL C00357 V=800.0 PL=0
MOVL C00358 V=800.0 PL=0
MOVL C00359 V=800.0 PL=0
MOVL C00360 V=800.0 PL=0
MOVL C00361 V=800.0 PL=0
MOVL C00362 V=800.0 PL=0
MOVL C00363 V=800.0 PL=0
MOVL C00364 V=800.0 PL=0
MOVL C00365 V=800.0 PL=0
MOVL C00366 V=800.0 PL=0
MOVL C00367 V=800.0 PL=0
MOVL C00368 V=800.0 PL=0
MOVL C00369 V=800.0 PL=0
MOVL C00370 V=800.0 PL=0
MOVL C00371 V=800.0 PL=0
MOVL C00372 V=800.0 PL=0
MOVL C00373 V=800.0 PL=0
MOVL C00374 V=800.0 PL=0
MOVL C00375 V=800.0 PL=0
MOVL C00376 V=800.0 PL=0
MOVL C00377 V=800.0 PL=0
MOVL C00378 V=800.0 PL=0
MOVL C00379 V=800.0 PL=0
MOVL C00380 V=800.0 PL=0
MOVL C00381 V=800.0 PL=0
MOVL C00382 V=800.0 PL=0
MOVL C00383 V=800.0 PL=0
MOVL C00384 V=800.0 PL=0
MOVL C00385 V=800.0 PL=0
MOVL C00386 V=800.0 PL=0
MOVL C00387 V=800.0 PL=0
MOVL C00388 V=800.0 PL=0
MOVL C00389 V=800.0 PL=0
MOVL C00390 V=800.0 PL=0
MOVL C00391 V=800.0 PL=0
MOVL C00392 V=800.0 PL=0
MOVL C00393 V=800.0 PL=0
MOVL C00394 V=800.0 PL=0
MOVL C00395 V=800.0 PL=0
MOVL C00396 V=800.0 PL=0
MOVL C00397 V=800.0 PL=0
MOVL C00398 V=800.0 PL=0
MOVL C00399 V=800.0 PL=0
MOVL C00400 V=800.0 PL=0
MOVL C00401 V=800.0 PL=0
MOVL C00402 V=800.0 PL=0
MOVL C00403 V=800.0 PL=0
MOVL C00404 V=800.0 PL=0
MOVL C00405 V=800.0 PL=0
MOVL C00406 V=800.0 PL=0
MOVL C00407 V=800.0 PL=0
MOVL C00408 V=800.0 PL=0
MOVL C00409 V=800.0 PL=0
MOVL C00410 V=800.0 PL=0
MOVL C00411 V=800.0 PL=0
MOVL C00412 V=800.0 PL=0
MOVL C00413 V=800.0 PL=0
MOVL C00414 V=800.0 PL=0
MOVL C00415 V=800.0 PL=0
MOVL C00416 V=800.0 PL=0
MOVL C00417 V=800.0 PL=0
MOVL C00418 V=800.0 PL=0
MOVL C00419 V=800.0 PL=0
MOVL C00420 V=800.0 PL=0
MOVL C00421 V=800.0 PL=0
MOVL C00422 V=800.0 PL=0
MOVL C00423 V=800.0 PL=0
MOVL C00424 V=800.0 PL=0
MOVL C00425 V=800.0 PL=0
MOVL C00426 V=800.0 PL=0
MOVL C00427 V=800.0 PL=0
MOVL C00428 V=800.0 PL=0
MOVL C00429 V=800.0 PL=0
MOVL C00430 V=800.0 PL=0
MOVL C00431 V=800.0 PL=0
MOVL C00432 V=800.0 PL=0
MOVL C00433 V=800.0 PL=0
MOVL C00434 V=800.0 PL=0
MOVL C00435 V=800.0 PL=0
MOVL C00436 V=800.0 PL=0
MOVL C00437 V=800.0 PL=0
MOVL C00438 V=800.0 PL=0
MOVL C00439 V=800.0 PL=0
MOVL C00440 V=800.0 PL=0
MOVL C00441 V=800.0 PL=0
MOVL C00442 V=800.0 PL=0
MOVL C00443 V=800.0 PL=0
MOVL C00444 V=800.0 PL=0
MOVL C00445 V=800.0 PL=0
MOVL C00446 V=800.0 PL=0
MOVL C00447 V=800.0 PL=0
MOVL C00448 V=800.0 PL=0
MOVL C00449 V=800.0 PL=0
MOVL C00450 V=800.0 PL=0
MOVL C00451 V=800.0 PL=0
MOVL C00452 V=800.0 PL=0
MOVL C00453 V=800.0 PL=0
MOVL C00454 V=800.0 PL=0
MOVL C00455 V=800.0 PL=0
MOVL C00456 V=800.0 PL=0
MOVL C00457 V=800.0 PL=0
MOVL C00458 V=800.0 PL=0
MOVL C00459 V=800.0 PL=0
MOVL C00460 V=800.0 PL=0
MOVL C00461 V=800.0 PL=0
MOVL C00462 V=800.0 PL=0
MOVL C00463 V=800.0 PL=0
MOVL C00464 V=800.0 PL=0
MOVL C00465 V=800.0 PL=0
MOVL C00466 V=800.0 PL=0
MOVL C00467 V=800.0 PL=0
MOVL C00468 V=800.0 PL=0
MOVL C00469 V=800.0 PL=0
MOVL C00470 V=800.0 PL=0
MOVL C00471 V=800.0 PL=0
MOVL C00472 V=800.0 PL=0
MOVL C00473 V=800.0 PL=0
MOVL C00474 V=800.0 PL=0
MOVL C00475 V=800.0 PL=0
MOVL C00476 V=800.0 PL=0
MOVL C00477 V=800.0 PL=0
MOVL C00478 V=800.0 PL=0
MOVL C00479 V=800.0 PL=0
MOVL C00480 V=800.0 PL=0
MOVL C00481 V=800.0 PL=0
MOVL C00482 V=800.0 PL=0
MOVL C00483 V=800.0 PL=0
MOVL C00484 V=800.0 PL=0
MOVL C00485 V=800.0 PL=0
MOVL C00486 V=800.0 PL=0
MOVL C00487 V=800.0 PL=0
MOVL C00488 V=800.0 PL=0
MOVL C00489 V=800.0 PL=0
MOVL C00490 V=800.0 PL=0
MOVL C00491 V=800.0 PL=0
MOVL C00492 V=800.0 PL=0
MOVL C00493 V=800.0 PL=0
MOVL C00494 V=800.0 PL=0
MOVL C00495 V=800.0 PL=0
MOVL C00496 V=800.0 PL=0
MOVL C00497 V=800.0 PL=0
MOVL C00498 V=800.0 PL=0
MOVL C00499 V=800.0 PL=0
MOVL C00500 V=800.0 PL=0
MOVL C00501 V=800.0 PL=0
MOVL C00502 V=800.0 PL=0
MOVL C00503 V=800.0 PL=0
MOVL C00504 V=800.0 PL=0
MOVL C00505 V=800.0 PL=0
MOVL C00506 V=800.0 PL=0
MOVL C00507 V=800.0 PL=0
MOVL C00508 V=800.0 PL=0
MOVL C00509 V=800.0 PL=0
MOVL C00510 V=800.0 PL=0
MOVL C00511 V=800.0 PL=0
MOVL C00512 V=800.0 PL=0
MOVL C00513 V=800.0 PL=0
MOVL C00514 V=800.0 PL=0
MOVL C00515 V=800.0 PL=0
MOVL C00516 V=800.0 PL=0
MOVL C00517 V=800.0 PL=0
MOVL C00518 V=800.0 PL=0
MOVL C00519 V=800.0 PL=0
MOVL C00520 V=800.0 PL=0
MOVL C00521 V=800.0 PL=0
MOVL C00522 V=800.0 PL=0
MOVL C00523 V=800.0 PL=0
MOVL C00524 V=800.0 PL=0
MOVL C00525 V=800.0 PL=0
MOVL C00526 V=800.0 PL=0
MOVL C00527 V=800.0 PL=0
MOVL C00528 V=800.0 PL=0
MOVL C00529 V=800.0 PL=0
MOVL C00530 V=800.0 PL=0
MOVL C00531 V=800.0 PL=0
MOVL C00532 V=800.0 PL=0
MOVL C00533 V=800.0 PL=0
MOVL C00534 V=800.0 PL=0
MOVL C00535 V=800.0 PL=0
MOVL C00536 V=800.0 PL=0
MOVL C00537 V=800.0 PL=0
MOVL C00538 V=800.0 PL=0
MOVL C00539 V=800.0 PL=0
MOVL C00540 V=800.0 PL=0
MOVL C00541 V=800.0 PL=0
MOVL C00542 V=800.0 PL=0
MOVL C00543 V=800.0 PL=0
MOVL C00544 V=800.0 PL=0
MOVL C00545 V=800.0 PL=0
MOVL C00546 V=800.0 PL=0
MOVL C00547 V=800.0 PL=0
MOVL C00548 V=800.0 PL=0
MOVL C00549 V=800.0 PL=0
MOVL C00550 V=800.0 PL=0
MOVL C00551 V=800.0 PL=0
MOVL C00552 V=800.0 PL=0
MOVL C00553 V=800.0 PL=0
MOVL C00554 V=800.0 PL=0
MOVL C00555 V=800.0 PL=0
MOVL C00556 V=800.0 PL=0
MOVL C00557 V=800.0 PL=0
MOVL C00558 V=800.0 PL=0
MOVL C00559 V=800.0 PL=0
MOVL C00560 V=800.0 PL=0
MOVL C00561 V=800.0 PL=0
MOVL C00562 V=800.0 PL=0
MOVL C00563 V=800.0 PL=0
MOVL C00564 V=800.0 PL=0
MOVL C00565 V=800.0 PL=0
MOVL C00566 V=800.0 PL=0
MOVL C00567 V=800.0 PL=0
MOVL C00568 V=800.0 PL=0
MOVL C00569 V=800.0 PL=0
MOVL C00570 V=800.0 PL=0
MOVL C00571 V=800.0 PL=0
MOVL C00572 V=800.0 PL=0
MOVL C00573 V=800.0 PL=0
MOVL C00574 V=800.0 PL=0
MOVL C00575 V=800.0 PL=0
MOVL C00576 V=800.0 PL=0
MOVL C00577 V=800.0 PL=0
MOVL C00578 V=800.0 PL=0
MOVL C00579 V=800.0 PL=0
MOVL C00580 V=800.0 PL=0
MOVL C00581 V=800.0 PL=0
MOVL C00582 V=800.0 PL=0
MOVL C00583 V=800.0 PL=0
MOVL C00584 V=800.0 PL=0
MOVL C00585 V=800.0 PL=0
MOVL C00586 V=800.0 PL=0
MOVL C00587 V=800.0 PL=0
MOVL C00588 V=800.0 PL=0
MOVL C00589 V=800.0 PL=0
MOVL C00590 V=800.0 PL=0
MOVL C00591 V=800.0 PL=0
MOVL C00592 V=800.0 PL=0
MOVL C00593 V=800.0 PL=0
MOVL C00594 V=800.0 PL=0
MOVL C00595 V=800.0 PL=0
MOVL C00596 V=800.0 PL=0
MOVL C00597 V=800.0 PL=0
MOVL C00598 V=800.0 PL=0
MOVL C00599 V=800.0 PL=0
MOVL C00600 V=800.0 PL=0
MOVL C00601 V=800.0 PL=0
MOVL C00602 V=800.0 PL=0
MOVL C00603 V=800.0 PL=0
MOVL C00604 V=800.0 PL=0
MOVL C00605 V=800.0 PL=0
MOVL C00606 V=800.0 PL=0
MOVL C00607 V=800.0 PL=0
MOVL C00608 V=800.0 PL=0
MOVL C00609 V=800.0 PL=0
MOVL C00610 V=800.0 PL=0
MOVL C00611 V=800.0 PL=0
MOVL C00612 V=800.0 PL=0
MOVL C00613 V=800.0 PL=0
MOVL C00614 V=800.0 PL=0
MOVL C00615 V=800.0 PL=0
MOVL C00616 V=800.0 PL=0
MOVL C00617 V=800.0 PL=0
MOVL C00618 V=800.0 PL=0
MOVL C00619 V=800.0 PL=0
MOVL C00620 V=800.0 PL=0
MOVL C00621 V=800.0 PL=0
MOVL C00622 V=800.0 PL=0
MOVL C00623 V=800.0 PL=0
MOVL C00624 V=800.0 PL=0
MOVL C00625 V=800.0 PL=0
MOVL C00626 V=800.0 PL=0
MOVL C00627 V=800.0 PL=0
MOVL C00628 V=800.0 PL=0
MOVL C00629 V=800.0 PL=0
MOVL C00630 V=800.0 PL=0
MOVL C00631 V=800.0 PL=0
MOVL C00632 V=800.0 PL=0
MOVL C00633 V=800.0 PL=0
MOVL C00634 V=800.0 PL=0
MOVL C00635 V=800.0 PL=0
MOVL C00636 V=800.0 PL=0
MOVL C00637 V=800.0 PL=0
MOVL C00638 V=800.0 PL=0
MOVL C00639 V=800.0 PL=0
MOVL C00640 V=800.0 PL=0
MOVL C00641 V=800.0 PL=0
MOVL C00642 V=800.0 PL=0
MOVL C00643 V=800.0 PL=0
MOVL C00644 V=800.0 PL=0
MOVL C00645 V=800.0 PL=0
MOVL C00646 V=800.0 PL=0
MOVL C00647 V=800.0 PL=0
MOVL C00648 V=800.0 PL=0
MOVL C00649 V=800.0 PL=0
MOVL C00650 V=800.0 PL=0
MOVL C00651 V=800.0 PL=0
MOVL C00652 V=800.0 PL=0
MOVL C00653 V=800.0 PL=0
MOVL C00654 V=800.0 PL=0
MOVL C00655 V=800.0 PL=0
MOVL C00656 V=800.0 PL=0
MOVL C00657 V=800.0 PL=0
MOVL C00658 V=800.0 PL=0
MOVL C00659 V=800.0 PL=0
MOVL C00660 V=800.0 PL=0
MOVL C00661 V=800.0 PL=0
MOVL C00662 V=800.0 PL=0
MOVL C00663 V=800.0 PL=0
MOVL C00664 V=800.0 PL=0
MOVL C00665 V=800.0 PL=0
MOVL C00666 V=800.0 PL=0
MOVL C00667 V=800.0 PL=0
MOVL C00668 V=800.0 PL=0
MOVL C00669 V=800.0 PL=0
MOVL C00670 V=800.0 PL=0
MOVL C00671 V=800.0 PL=0
MOVL C00672 V=800.0 PL=0
MOVL C00673 V=800.0 PL=0
MOVL C00674 V=800.0 PL=0
MOVL C00675 V=800.0 PL=0
MOVL C00676 V=800.0 PL=0
MOVL C00677 V=800.0 PL=0
MOVL C00678 V=800.0 PL=0
MOVL C00679 V=800.0 PL=0
MOVL C00680 V=800.0 PL=0
MOVL C00681 V=800.0 PL=0
MOVL C00682 V=800.0 PL=0
MOVL C00683 V=800.0 PL=0
MOVL C00684 V=800.0 PL=0
MOVL C00685 V=800.0 PL=0
MOVL C00686 V=800.0 PL=0
MOVL C00687 V=800.0 PL=0
MOVL C00688 V=800.0 PL=0
MOVL C00689 V=800.0 PL=0
MOVL C00690 V=800.0 PL=0
MOVL C00691 V=800.0 PL=0
MOVL C00692 V=800.0 PL=0
MOVL C00693 V=800.0 PL=0
MOVL C00694 V=800.0 PL=0
MOVL C00695 V=800.0 PL=0
MOVL C00696 V=800.0 PL=0
MOVL C00697 V=800.0 PL=0
MOVL C00698 V=800.0 PL=0
MOVL C00699 V=800.0 PL=0
MOVL C00700 V=800.0 PL=0
MOVL C00701 V=800.0 PL=0
MOVL C00702 V=800.0 PL=0
MOVL C00703 V=800.0 PL=0
MOVL C00704 V=800.0 PL=0
MOVL C00705 V=800.0 PL=0
MOVL C00706 V=800.0 PL=0
MOVL C00707 V=800.0 PL=0
MOVL C00708 V=800.0 PL=0
MOVL C00709 V=800.0 PL=0
MOVL C00710 V=800.0 PL=0
MOVL C00711 V=800.0 PL=0
MOVL C00712 V=800.0 PL=0
MOVL C00713 V=800.0 PL=0
MOVL C00714 V=800.0 PL=0
MOVL C00715 V=800.0 PL=0
MOVL C00716 V=800.0 PL=0
MOVL C00717 V=800.0 PL=0
MOVL C00718 V=800.0 PL=0
MOVL C00719 V=800.0 PL=0
MOVL C00720 V=800.0 PL=0
MOVL C00721 V=800.0 PL=0
MOVL C00722 V=800.0 PL=0
MOVL C00723 V=800.0 PL=0
MOVL C00724 V=800.0 PL=0
MOVL C00725 V=800.0 PL=0
MOVL C00726 V=800.0 PL=0
MOVL C00727 V=800.0 PL=0
MOVL C00728 V=800.0 PL=0
MOVL C00729 V=800.0 PL=0
MOVL C00730 V=800.0 PL=0
MOVL C00731 V=800.0 PL=0
MOVL C00732 V=800.0 PL=0
MOVL C00733 V=800.0 PL=0
MOVL C00734 V=800.0 PL=0
MOVL C00735 V=800.0 PL=0
MOVL C00736 V=800.0 PL=0
MOVL C00737 V=800.0 PL=0
MOVL C00738 V=800.0 PL=0
MOVL C00739 V=800.0 PL=0
MOVL C00740 V=800.0 PL=0
MOVL C00741 V=800.0 PL=0
MOVL C00742 V=800.0 PL=0
MOVL C00743 V=800.0 PL=0
MOVL C00744 V=800.0 PL=0
MOVL C00745 V=800.0 PL=0
MOVL C00746 V=800.0 PL=0
MOVL C00747 V=800.0 PL=0
MOVL C00748 V=800.0 PL=0
MOVL C00749 V=800.0 PL=0
MOVL C00750 V=800.0 PL=0
MOVL C00751 V=800.0 PL=0
MOVL C00752 V=800.0 PL=0
MOVL C00753 V=800.0 PL=0
MOVL C00754 V=800.0 PL=0
MOVL C00755 V=800.0 PL=0
MOVL C00756 V=800.0 PL=0
MOVL C00757 V=800.0 PL=0
MOVL C00758 V=800.0 PL=0
MOVL C00759 V=800.0 PL=0
MOVL C00760 V=800.0 PL=0
MOVL C00761 V=800.0 PL=0
MOVL C00762 V=800.0 PL=0
MOVL C00763 V=800.0 PL=0
MOVL C00764 V=800.0 PL=0
MOVL C00765 V=800.0 PL=0
MOVL C00766 V=800.0 PL=0
MOVL C00767 V=800.0 PL=0
MOVL C00768 V=800.0 PL=0
MOVL C00769 V=800.0 PL=0
MOVL C00770 V=800.0 PL=0
MOVL C00771 V=800.0 PL=0
MOVL C00772 V=800.0 PL=0
MOVL C00773 V=800.0 PL=0
MOVL C00774 V=800.0 PL=0
MOVL C00775 V=800.0 PL=0
MOVL C00776 V=800.0 PL=0
MOVL C00777 V=800.0 PL=0
MOVL C00778 V=800.0 PL=0
MOVL C00779 V=800.0 PL=0
MOVL C00780 V=800.0 PL=0
MOVL C00781 V=800.0 PL=0
MOVL C00782 V=800.0 PL=0
MOVL C00783 V=800.0 PL=0
MOVL C00784 V=800.0 PL=0
MOVL C00785 V=800.0 PL=0
MOVL C00786 V=800.0 PL=0
MOVL C00787 V=800.0 PL=0
MOVL C00788 V=800.0 PL=0
MOVL C00789 V=800.0 PL=0
MOVL C00790 V=800.0 PL=0
MOVL C00791 V=800.0 PL=0
MOVL C00792 V=800.0 PL=0
MOVL C00793 V=800.0 PL=0
MOVL C00794 V=800.0 PL=0
MOVL C00795 V=800.0 PL=0
MOVL C00796 V=800.0 PL=0
MOVL C00797 V=800.0 PL=0
MOVL C00798 V=800.0 PL=0
MOVL C00799 V=800.0 PL=0
MOVL C00800 V=800.0 PL=0
MOVL C00801 V=800.0 PL=0
MOVL C00802 V=800.0 PL=0
MOVL C00803 V=800.0 PL=0
MOVL C00804 V=800.0 PL=0
MOVL C00805 V=800.0 PL=0
MOVL C00806 V=800.0 PL=0
MOVL C00807 V=800.0 PL=0
MOVL C00808 V=800.0 PL=0
MOVL C00809 V=800.0 PL=0
MOVL C00810 V=800.0 PL=0
MOVL C00811 V=800.0 PL=0
MOVL C00812 V=800.0 PL=0
MOVL C00813 V=800.0 PL=0
MOVL C00814 V=800.0 PL=0
MOVL C00815 V=800.0 PL=0
MOVL C00816 V=800.0 PL=0
MOVL C00817 V=800.0 PL=0
MOVL C00818 V=800.0 PL=0
MOVL C00819 V=800.0 PL=0
MOVL C00820 V=800.0 PL=0
MOVL C00821 V=800.0 PL=0
MOVL C00822 V=800.0 PL=0
MOVL C00823 V=800.0 PL=0
MOVL C00824 V=800.0 PL=0
MOVL C00825 V=800.0 PL=0
MOVL C00826 V=800.0 PL=0
MOVL C00827 V=800.0 PL=0
MOVL C00828 V=800.0 PL=0
MOVL C00829 V=800.0 PL=0
MOVL C00830 V=800.0 PL=0
MOVL C00831 V=800.0 PL=0
MOVL C00832 V=800.0 PL=0
MOVL C00833 V=800.0 PL=0
MOVL C00834 V=800.0 PL=0
MOVL C00835 V=800.0 PL=0
MOVL C00836 V=800.0 PL=0
MOVL C00837 V=800.0 PL=0
MOVL C00838 V=800.0 PL=0
MOVL C00839 V=800.0 PL=0
MOVL C00840 V=800.0 PL=0
MOVL C00841 V=800.0 PL=0
MOVL C00842 V=800.0 PL=0
MOVL C00843 V=800.0 PL=0
MOVL C00844 V=800.0 PL=0
MOVL C00845 V=800.0 PL=0
MOVL C00846 V=800.0 PL=0
MOVL C00847 V=800.0 PL=0
MOVL C00848 V=800.0 PL=0
MOVL C00849 V=800.0 PL=0
MOVL C00850 V=800.0 PL=0
MOVL C00851 V=800.0 PL=0
MOVL C00852 V=800.0 PL=0
MOVL C00853 V=800.0 PL=0
MOVL C00854 V=800.0 PL=0
MOVL C00855 V=800.0 PL=0
MOVL C00856 V=800.0 PL=0
MOVL C00857 V=800.0 PL=0
MOVL C00858 V=800.0 PL=0
MOVL C00859 V=800.0 PL=0
MOVL C00860 V=800.0 PL=0
MOVL C00861 V=800.0 PL=0
MOVL C00862 V=800.0 PL=0
MOVL C00863 V=800.0 PL=0
MOVL C00864 V=800.0 PL=0
MOVL C00865 V=800.0 PL=0
MOVL C00866 V=800.0 PL=0
MOVL C00867 V=800.0 PL=0
MOVL C00868 V=800.0 PL=0
MOVL C00869 V=800.0 PL=0
MOVL C00870 V=800.0 PL=0
MOVL C00871 V=800.0 PL=0
MOVL C00872 V=800.0 PL=0
MOVL C00873 V=800.0 PL=0
MOVL C00874 V=800.0 PL=0
MOVL C00875 V=800.0 PL=0
MOVL C00876 V=800.0 PL=0
MOVL C00877 V=800.0 PL=0
MOVL C00878 V=800.0 PL=0
MOVL C00879 V=800.0 PL=0
MOVL C00880 V=800.0 PL=0
MOVL C00881 V=800.0 PL=0
MOVL C00882 V=800.0 PL=0
MOVL C00883 V=800.0 PL=0
MOVL C00884 V=800.0 PL=0
MOVL C00885 V=800.0 PL=0
MOVL C00886 V=800.0 PL=0
MOVL C00887 V=800.0 PL=0
MOVL C00888 V=800.0 PL=0
MOVL C00889 V=800.0 PL=0
MOVL C00890 V=800.0 PL=0
MOVL C00891 V=800.0 PL=0
MOVL C00892 V=800.0 PL=0
MOVL C00893 V=800.0 PL=0
MOVL C00894 V=800.0 PL=0
MOVL C00895 V=800.0 PL=0
MOVL C00896 V=800.0 PL=0
MOVL C00897 V=800.0 PL=0
MOVL C00898 V=800.0 PL=0
MOVL C00899 V=800.0 PL=0
MOVL C00900 V=800.0 PL=0
MOVL C00901 V=800.0 PL=0
MOVL C00902 V=800.0 PL=0
MOVL C00903 V=800.0 PL=0
MOVL C00904 V=800.0 PL=0
MOVL C00905 V=800.0 PL=0
MOVL C00906 V=800.0 PL=0
MOVL C00907 V=800.0 PL=0
MOVL C00908 V=800.0 PL=0
MOVL C00909 V=800.0 PL=0
MOVL C00910 V=800.0 PL=0
MOVL C00911 V=800.0 PL=0
MOVL C00912 V=800.0 PL=0
MOVL C00913 V=800.0 PL=0
MOVL C00914 V=800.0 PL=0
MOVL C00915 V=800.0 PL=0
MOVL C00916 V=800.0 PL=0
MOVL C00917 V=800.0 PL=0
MOVL C00918 V=800.0 PL=0
MOVL C00919 V=800.0 PL=0
MOVL C00920 V=800.0 PL=0
MOVL C00921 V=800.0 PL=0
MOVL C00922 V=800.0 PL=0
MOVL C00923 V=800.0 PL=0
MOVL C00924 V=800.0 PL=0
MOVL C00925 V=800.0 PL=0
MOVL C00926 V=800.0 PL=0
MOVL C00927 V=800.0 PL=0
MOVL C00928 V=800.0 PL=0
MOVL C00929 V=800.0 PL=0
MOVL C00930 V=800.0 PL=0
MOVL C00931 V=800.0 PL=0
MOVL C00932 V=800.0 PL=0
MOVL C00933 V=800.0 PL=0
MOVL C00934 V=800.0 PL=0
MOVL C00935 V=800.0 PL=0
MOVL C00936 V=800.0 PL=0
MOVL C00937 V=800.0 PL=0
MOVL C00938 V=800.0 PL=0
MOVL C00939 V=800.0 PL=0
MOVL C00940 V=800.0 PL=0
MOVL C00941 V=800.0 PL=0
MOVL C00942 V=800.0 PL=0
MOVL C00943 V=800.0 PL=0
MOVL C00944 V=800.0 PL=0
MOVL C00945 V=800.0 PL=0
MOVL C00946 V=800.0 PL=0
MOVL C00947 V=800.0 PL=0
MOVL C00948 V=800.0 PL=0
MOVL C00949 V=800.0 PL=0
MOVL C00950 V=800.0 PL=0
MOVL C00951 V=800.0 PL=0
MOVL C00952 V=800.0 PL=0
MOVL C00953 V=800.0 PL=0
MOVL C00954 V=800.0 PL=0
MOVL C00955 V=800.0 PL=0
MOVL C00956 V=800.0 PL=0
MOVL C00957 V=800.0 PL=0
MOVL C00958 V=800.0 PL=0
MOVL C00959 V=800.0 PL=0
MOVL C00960 V=800.0 PL=0
MOVL C00961 V=800.0 PL=0
MOVL C00962 V=800.0 PL=0
MOVL C00963 V=800.0 PL=0
MOVL C00964 V=800.0 PL=0
MOVL C00965 V=800.0 PL=0
MOVL C00966 V=800.0 PL=0
MOVL C00967 V=800.0 PL=0
MOVL C00968 V=800.0 PL=0
MOVL C00969 V=800.0 PL=0
MOVL C00970 V=800.0 PL=0
MOVL C00971 V=800.0 PL=0
MOVL C00972 V=800.0 PL=0
MOVL C00973 V=800.0 PL=0
MOVL C00974 V=800.0 PL=0
MOVL C00975 V=800.0 PL=0
MOVL C00976 V=800.0 PL=0
MOVL C00977 V=800.0 PL=0
MOVL C00978 V=800.0 PL=0
MOVL C00979 V=800.0 PL=0
MOVL C00980 V=800.0 PL=0
MOVL C00981 V=800.0 PL=0
MOVL C00982 V=800.0 PL=0
MOVL C00983 V=800.0 PL=0
MOVL C00984 V=800.0 PL=0
MOVL C00985 V=800.0 PL=0
MOVL C00986 V=800.0 PL=0
MOVL C00987 V=800.0 PL=0
MOVL C00988 V=800.0 PL=0
MOVL C00989 V=800.0 PL=0
MOVL C00990 V=800.0 PL=0
MOVL C00991 V=800.0 PL=0
MOVL C00992 V=800.0 PL=0
MOVL C00993 V=800.0 PL=0
MOVL C00994 V=800.0 PL=0
MOVL C00995 V=800.0 PL=0
MOVL C00996 V=800.0 PL=0
MOVL C00997 V=800.0 PL=0
MOVL C00998 V=800.0 PL=0
MOVL C00999 V=800.0 PL=0
MOVL C01000 V=800.0 PL=0
MOVL C01001 V=800.0 PL=0
MOVL C01002 V=800.0 PL=0
MOVL C01003 V=800.0 PL=0
MOVL C01004 V=800.0 PL=0
MOVL C01005 V=800.0 PL=0
MOVL C01006 V=800.0 PL=0
MOVL C01007 V=800.0 PL=0
MOVL C01008 V=800.0 PL=0
MOVL C01009 V=800.0 PL=0
MOVL C01010 V=800.0 PL=0
MOVL C01011 V=800.0 PL=0
MOVL C01012 V=800.0 PL=0
MOVL C01013 V=800.0 PL=0
MOVL C01014 V=800.0 PL=0
MOVL C01015 V=800.0 PL=0
MOVL C01016 V=800.0 PL=0
MOVL C01017 V=800.0 PL=0
MOVL C01018 V=800.0 PL=0
MOVL C01019 V=800.0 PL=0
MOVL C01020 V=800.0 PL=0
MOVL C01021 V=800.0 PL=0
MOVL C01022 V=800.0 PL=0
MOVL C01023 V=800.0 PL=0
MOVL C01024 V=800.0 PL=0
MOVL C01025 V=800.0 PL=0
MOVL C01026 V=800.0 PL=0
MOVL C01027 V=800.0 PL=0
MOVL C01028 V=800.0 PL=0
MOVL C01029 V=800.0 PL=0
MOVL C01030 V=800.0 PL=0
MOVL C01031 V=800.0 PL=0
MOVL C01032 V=800.0 PL=0
MOVL C01033 V=800.0 PL=0
MOVL C01034 V=800.0 PL=0
MOVL C01035 V=800.0 PL=0
MOVL C01036 V=800.0 PL=0
MOVL C01037 V=800.0 PL=0
MOVL C01038 V=800.0 PL=0
MOVL C01039 V=800.0 PL=0
MOVL C01040 V=800.0 PL=0
MOVL C01041 V=800.0 PL=0
MOVL C01042 V=800.0 PL=0
MOVL C01043 V=800.0 PL=0
MOVL C01044 V=800.0 PL=0
MOVL C01045 V=800.0 PL=0
MOVL C01046 V=800.0 PL=0
MOVL C01047 V=800.0 PL=0
MOVL C01048 V=800.0 PL=0
MOVL C01049 V=800.0 PL=0
MOVL C01050 V=800.0 PL=0
MOVL C01051 V=800.0 PL=0
MOVL C01052 V=800.0 PL=0
MOVL C01053 V=800.0 PL=0
MOVL C01054 V=800.0 PL=0
MOVL C01055 V=800.0 PL=0
MOVL C01056 V=800.0 PL=0
MOVL C01057 V=800.0 PL=0
MOVL C01058 V=800.0 PL=0
MOVL C01059 V=800.0 PL=0
MOVL C01060 V=800.0 PL=0
MOVL C01061 V=800.0 PL=0
MOVL C01062 V=800.0 PL=0
MOVL C01063 V=800.0 PL=0
MOVL C01064 V=800.0 PL=0
MOVL C01065 V=800.0 PL=0
MOVL C01066 V=800.0 PL=0
MOVL C01067 V=800.0 PL=0
MOVL C01068 V=800.0 PL=0
MOVL C01069 V=800.0 PL=0
MOVL C01070 V=800.0 PL=0
MOVL C01071 V=800.0 PL=0
MOVL C01072 V=800.0 PL=0
MOVL C01073 V=800.0 PL=0
MOVL C01074 V=800.0 PL=0
MOVL C01075 V=800.0 PL=0
MOVL C01076 V=800.0 PL=0
MOVL C01077 V=800.0 PL=0
MOVL C01078 V=800.0 PL=0
MOVL C01079 V=800.0 PL=0
MOVL C01080 V=800.0 PL=0
MOVL C01081 V=800.0 PL=0
MOVL C01082 V=800.0 PL=0
MOVL C01083 V=800.0 PL=0
MOVL C01084 V=800.0 PL=0
MOVL C01085 V=800.0 PL=0
MOVL C01086 V=800.0 PL=0
MOVL C01087 V=800.0 PL=0
MOVL C01088 V=800.0 PL=0
MOVL C01089 V=800.0 PL=0
MOVL C01090 V=800.0 PL=0
MOVL C01091 V=800.0 PL=0
MOVL C01092 V=800.0 PL=0
MOVL C01093 V=800.0 PL=0
MOVL C01094 V=800.0 PL=0
MOVL C01095 V=800.0 PL=0
MOVL C01096 V=800.0 PL=0
MOVL C01097 V=800.0 PL=0
MOVL C01098 V=800.0 PL=0
MOVL C01099 V=800.0 PL=0
MOVL C01100 V=800.0 PL=0
MOVL C01101 V=800.0 PL=0
MOVL C01102 V=800.0 PL=0
MOVL C01103 V=800.0 PL=0
MOVL C01104 V=800.0 PL=0
MOVL C01105 V=800.0 PL=0
MOVL C01106 V=800.0 PL=0
MOVL C01107 V=800.0 PL=0
MOVL C01108 V=800.0 PL=0
MOVL C01109 V=800.0 PL=0
MOVL C01110 V=800.0 PL=0
MOVL C01111 V=800.0 PL=0
MOVL C01112 V=800.0 PL=0
MOVL C01113 V=800.0 PL=0
MOVL C01114 V=800.0 PL=0
MOVL C01115 V=800.0 PL=0
MOVL C01116 V=800.0 PL=0
MOVL C01117 V=800.0 PL=0
MOVL C01118 V=800.0 PL=0
MOVL C01119 V=800.0 PL=0
MOVL C01120 V=800.0 PL=0
MOVL C01121 V=800.0 PL=0
MOVL C01122 V=800.0 PL=0
MOVL C01123 V=800.0 PL=0
MOVL C01124 V=800.0 PL=0
MOVL C01125 V=800.0 PL=0
MOVL C01126 V=800.0 PL=0
MOVL C01127 V=800.0 PL=0
MOVL C01128 V=800.0 PL=0
MOVL C01129 V=800.0 PL=0
MOVL C01130 V=800.0 PL=0
MOVL C01131 V=800.0 PL=0
MOVL C01132 V=800.0 PL=0
MOVL C01133 V=800.0 PL=0
MOVL C01134 V=800.0 PL=0
MOVL C01135 V=800.0 PL=0
MOVL C01136 V=800.0 PL=0
MOVL C01137 V=800.0 PL=0
MOVL C01138 V=800.0 PL=0
MOVL C01139 V=800.0 PL=0
MOVL C01140 V=800.0 PL=0
MOVL C01141 V=800.0 PL=0
MOVL C01142 V=800.0 PL=0
MOVL C01143 V=800.0 PL=0
MOVL C01144 V=800.0 PL=0
MOVL C01145 V=800.0 PL=0
MOVL C01146 V=800.0 PL=0
MOVL C01147 V=800.0 PL=0
MOVL C01148 V=800.0 PL=0
MOVL C01149 V=800.0 PL=0
MOVL C01150 V=800.0 PL=0
MOVL C01151 V=800.0 PL=0
MOVL C01152 V=800.0 PL=0
MOVL C01153 V=800.0 PL=0
MOVL C01154 V=800.0 PL=0
MOVL C01155 V=800.0 PL=0
MOVL C01156 V=800.0 PL=0
MOVL C01157 V=800.0 PL=0
MOVL C01158 V=800.0 PL=0
MOVL C01159 V=800.0 PL=0
MOVL C01160 V=800.0 PL=0
MOVL C01161 V=800.0 PL=0
MOVL C01162 V=800.0 PL=0
MOVL C01163 V=800.0 PL=0
MOVL C01164 V=800.0 PL=0
MOVL C01165 V=800.0 PL=0
MOVL C01166 V=800.0 PL=0
MOVL C01167 V=800.0 PL=0
MOVL C01168 V=800.0 PL=0
MOVL C01169 V=800.0 PL=0
MOVL C01170 V=800.0 PL=0
MOVL C01171 V=800.0 PL=0
MOVL C01172 V=800.0 PL=0
MOVL C01173 V=800.0 PL=0
MOVL C01174 V=800.0 PL=0
MOVL C01175 V=800.0 PL=0
MOVL C01176 V=800.0 PL=0
MOVL C01177 V=800.0 PL=0
MOVL C01178 V=800.0 PL=0
MOVL C01179 V=800.0 PL=0
MOVL C01180 V=800.0 PL=0
MOVL C01181 V=800.0 PL=0
MOVL C01182 V=800.0 PL=0
MOVL C01183 V=800.0 PL=0
MOVL C01184 V=800.0 PL=0
MOVL C01185 V=800.0 PL=0
MOVL C01186 V=800.0 PL=0
MOVL C01187 V=800.0 PL=0
MOVL C01188 V=800.0 PL=0
MOVL C01189 V=800.0 PL=0
MOVL C01190 V=800.0 PL=0
MOVL C01191 V=800.0 PL=0
MOVL C01192 V=800.0 PL=0
MOVL C01193 V=800.0 PL=0
MOVL C01194 V=800.0 PL=0
MOVL C01195 V=800.0 PL=0
MOVL C01196 V=800.0 PL=0
MOVL C01197 V=800.0 PL=0
MOVL C01198 V=800.0 PL=0
MOVL C01199 V=800.0 PL=0
MOVL C01200 V=800.0 PL=0
MOVL C01201 V=800.0 PL=0
MOVL C01202 V=800.0 PL=0
MOVL C01203 V=800.0 PL=0
MOVL C01204 V=800.0 PL=0
MOVL C01205 V=800.0 PL=0
MOVL C01206 V=800.0 PL=0
MOVL C01207 V=800.0 PL=0
MOVL C01208 V=800.0 PL=0
MOVL C01209 V=800.0 PL=0
MOVL C01210 V=800.0 PL=0
MOVL C01211 V=800.0 PL=0
MOVL C01212 V=800.0 PL=0
MOVL C01213 V=800.0 PL=0
MOVL C01214 V=800.0 PL=0
MOVL C01215 V=800.0 PL=0
MOVL C01216 V=800.0 PL=0
MOVL C01217 V=800.0 PL=0
MOVL C01218 V=800.0 PL=0
MOVL C01219 V=800.0 PL=0
MOVL C01220 V=800.0 PL=0
MOVL C01221 V=800.0 PL=0
MOVL C01222 V=800.0 PL=0
MOVL C01223 V=800.0 PL=0
MOVL C01224 V=800.0 PL=0
MOVL C01225 V=800.0 PL=0
MOVL C01226 V=800.0 PL=0
MOVL C01227 V=800.0 PL=0
MOVL C01228 V=800.0 PL=0
MOVL C01229 V=800.0 PL=0
MOVL C01230 V=800.0 PL=0
MOVL C01231 V=800.0 PL=0
MOVL C01232 V=800.0 PL=0
MOVL C01233 V=800.0 PL=0
MOVL C01234 V=800.0 PL=0
MOVL C01235 V=800.0 PL=0
MOVL C01236 V=800.0 PL=0
MOVL C01237 V=800.0 PL=0
MOVL C01238 V=800.0 PL=0
MOVL C01239 V=800.0 PL=0
MOVL C01240 V=800.0 PL=0
MOVL C01241 V=800.0 PL=0
MOVL C01242 V=800.0 PL=0
MOVL C01243 V=800.0 PL=0
MOVL C01244 V=800.0 PL=0
MOVL C01245 V=800.0 PL=0
MOVL C01246 V=800.0 PL=0
MOVL C01247 V=800.0 PL=0
MOVL C01248 V=800.0 PL=0
MOVL C01249 V=800.0 PL=0
MOVL C01250 V=800.0 PL=0
MOVL C01251 V=800.0 PL=0
MOVL C01252 V=800.0 PL=0
MOVL C01253 V=800.0 PL=0
MOVL C01254 V=800.0 PL=0
MOVL C01255 V=800.0 PL=0
MOVL C01256 V=800.0 PL=0
MOVL C01257 V=800.0 PL=0
MOVL C01258 V=800.0 PL=0
MOVL C01259 V=800.0 PL=0
MOVL C01260 V=800.0 PL=0
MOVL C01261 V=800.0 PL=0
MOVL C01262 V=800.0 PL=0
MOVL C01263 V=800.0 PL=0
MOVL C01264 V=800.0 PL=0
MOVL C01265 V=800.0 PL=0
MOVL C01266 V=800.0 PL=0
MOVL C01267 V=800.0 PL=0
MOVL C01268 V=800.0 PL=0
MOVL C01269 V=800.0 PL=0
MOVL C01270 V=800.0 PL=0
MOVL C01271 V=800.0 PL=0
MOVL C01272 V=800.0 PL=0
MOVL C01273 V=800.0 PL=0
MOVL C01274 V=800.0 PL=0
MOVL C01275 V=800.0 PL=0
MOVL C01276 V=800.0 PL=0
MOVL C01277 V=800.0 PL=0
MOVL C01278 V=800.0 PL=0
MOVL C01279 V=800.0 PL=0
MOVL C01280 V=800.0 PL=0
MOVL C01281 V=800.0 PL=0
MOVL C01282 V=800.0 PL=0
MOVL C01283 V=800.0 PL=0
MOVL C01284 V=800.0 PL=0
MOVL C01285 V=800.0 PL=0
MOVL C01286 V=800.0 PL=0
MOVL C01287 V=800.0 PL=0
MOVL C01288 V=800.0 PL=0
MOVL C01289 V=800.0 PL=0
MOVL C01290 V=800.0 PL=0
MOVL C01291 V=800.0 PL=0
MOVL C01292 V=800.0 PL=0
MOVL C01293 V=800.0 PL=0
MOVL C01294 V=800.0 PL=0
MOVL C01295 V=800.0 PL=0
MOVL C01296 V=800.0 PL=0
MOVL C01297 V=800.0 PL=0
MOVL C01298 V=800.0 PL=0
MOVL C01299 V=800.0 PL=0
MOVL C01300 V=800.0 PL=0
MOVL C01301 V=800.0 PL=0
MOVL C01302 V=800.0 PL=0
MOVL C01303 V=800.0 PL=0
MOVL C01304 V=800.0 PL=0
MOVL C01305 V=800.0 PL=0
MOVL C01306 V=800.0 PL=0
MOVL C01307 V=800.0 PL=0
MOVL C01308 V=800.0 PL=0
MOVL C01309 V=800.0 PL=0
MOVL C01310 V=800.0 PL=0
MOVL C01311 V=800.0 PL=0
MOVL C01312 V=800.0 PL=0
MOVL C01313 V=800.0 PL=0
MOVL C01314 V=800.0 PL=0
MOVL C01315 V=800.0 PL=0
MOVL C01316 V=800.0 PL=0
MOVL C01317 V=800.0 PL=0
MOVL C01318 V=800.0 PL=0
MOVL C01319 V=800.0 PL=0
MOVL C01320 V=800.0 PL=0
MOVL C01321 V=800.0 PL=0
MOVL C01322 V=800.0 PL=0
MOVL C01323 V=800.0 PL=0
MOVL C01324 V=800.0 PL=0
MOVL C01325 V=800.0 PL=0
MOVL C01326 V=800.0 PL=0
MOVL C01327 V=800.0 PL=0
MOVL C01328 V=800.0 PL=0
MOVL C01329 V=800.0 PL=0
MOVL C01330 V=800.0 PL=0
MOVL C01331 V=800.0 PL=0
MOVL C01332 V=800.0 PL=0
MOVL C01333 V=800.0 PL=0
MOVL C01334 V=800.0 PL=0
MOVL C01335 V=800.0 PL=0
MOVL C01336 V=800.0 PL=0
MOVL C01337 V=800.0 PL=0
MOVL C01338 V=800.0 PL=0
MOVL C01339 V=800.0 PL=0
MOVL C01340 V=800.0 PL=0
MOVL C01341 V=800.0 PL=0
MOVL C01342 V=800.0 PL=0
MOVL C01343 V=800.0 PL=0
MOVL C01344 V=800.0 PL=0
MOVL C01345 V=800.0 PL=0
MOVL C01346 V=800.0 PL=0
MOVL C01347 V=800.0 PL=0
MOVL C01348 V=800.0 PL=0
MOVL C01349 V=800.0 PL=0
MOVL C01350 V=800.0 PL=0
MOVL C01351 V=800.0 PL=0
MOVL C01352 V=800.0 PL=0
MOVL C01353 V=800.0 PL=0
MOVL C01354 V=800.0 PL=0
MOVL C01355 V=800.0 PL=0
MOVL C01356 V=800.0 PL=0
MOVL C01357 V=800.0 PL=0
MOVL C01358 V=800.0 PL=0
MOVL C01359 V=800.0 PL=0
MOVL C01360 V=800.0 PL=0
MOVL C01361 V=800.0 PL=0
MOVL C01362 V=800.0 PL=0
MOVL C01363 V=800.0 PL=0
MOVL C01364 V=800.0 PL=0
MOVL C01365 V=800.0 PL=0
MOVL C01366 V=800.0 PL=0
MOVL C01367 V=800.0 PL=0
MOVL C01368 V=800.0 PL=0
MOVL C01369 V=800.0 PL=0
MOVL C01370 V=800.0 PL=0
MOVL C01371 V=800.0 PL=0
MOVL C01372 V=800.0 PL=0
MOVL C01373 V=800.0 PL=0
MOVL C01374 V=800.0 PL=0
MOVL C01375 V=800.0 PL=0
MOVL C01376 V=800.0 PL=0
MOVL C01377 V=800.0 PL=0
MOVL C01378 V=800.0 PL=0
MOVL C01379 V=800.0 PL=0
MOVL C01380 V=800.0 PL=0
MOVL C01381 V=800.0 PL=0
MOVL C01382 V=800.0 PL=0
MOVL C01383 V=800.0 PL=0
MOVL C01384 V=800.0 PL=0
MOVL C01385 V=800.0 PL=0
MOVL C01386 V=800.0 PL=0
MOVL C01387 V=800.0 PL=0
MOVL C01388 V=800.0 PL=0
MOVL C01389 V=800.0 PL=0
MOVL C01390 V=800.0 PL=0
MOVL C01391 V=800.0 PL=0
MOVL C01392 V=800.0 PL=0
MOVL C01393 V=800.0 PL=0
MOVL C01394 V=800.0 PL=0
MOVL C01395 V=800.0 PL=0
MOVL C01396 V=800.0 PL=0
MOVL C01397 V=800.0 PL=0
MOVL C01398 V=800.0 PL=0
MOVL C01399 V=800.0 PL=0
MOVL C01400 V=800.0 PL=0
MOVL C01401 V=800.0 PL=0
MOVL C01402 V=800.0 PL=0
MOVL C01403 V=800.0 PL=0
MOVL C01404 V=800.0 PL=0
MOVL C01405 V=800.0 PL=0
MOVL C01406 V=800.0 PL=0
MOVL C01407 V=800.0 PL=0
MOVL C01408 V=800.0 PL=0
MOVL C01409 V=800.0 PL=0
MOVL C01410 V=800.0 PL=0
MOVL C01411 V=800.0 PL=0
MOVL C01412 V=800.0 PL=0
MOVL C01413 V=800.0 PL=0
MOVL C01414 V=800.0 PL=0
MOVL C01415 V=800.0 PL=0
MOVL C01416 V=800.0 PL=0
MOVL C01417 V=800.0 PL=0
MOVL C01418 V=800.0 PL=0
MOVL C01419 V=800.0 PL=0
MOVL C01420 V=800.0 PL=0
MOVL C01421 V=800.0 PL=0
MOVL C01422 V=800.0 PL=0
MOVL C01423 V=800.0 PL=0
MOVL C01424 V=800.0 PL=0
MOVL C01425 V=800.0 PL=0
MOVL C01426 V=800.0 PL=0
MOVL C01427 V=800.0 PL=0
MOVL C01428 V=800.0 PL=0
MOVL C01429 V=800.0 PL=0
MOVL C01430 V=800.0 PL=0
MOVL C01431 V=800.0 PL=0
MOVL C01432 V=800.0 PL=0
MOVL C01433 V=800.0 PL=0
MOVL C01434 V=800.0 PL=0
MOVL C01435 V=800.0 PL=0
MOVL C01436 V=800.0 PL=0
MOVL C01437 V=800.0 PL=0
MOVL C01438 V=800.0 PL=0
MOVL C01439 V=800.0 PL=0
MOVL C01440 V=800.0 PL=0
MOVL C01441 V=800.0 PL=0
MOVL C01442 V=800.0 PL=0
MOVL C01443 V=800.0 PL=0
MOVL C01444 V=800.0 PL=0
MOVL C01445 V=800.0 PL=0
MOVL C01446 V=800.0 PL=0
MOVL C01447 V=800.0 PL=0
MOVL C01448 V=800.0 PL=0
MOVL C01449 V=800.0 PL=0
MOVL C01450 V=800.0 PL=0
MOVL C01451 V=800.0 PL=0
MOVL C01452 V=800.0 PL=0
MOVL C01453 V=800.0 PL=0
MOVL C01454 V=800.0 PL=0
MOVL C01455 V=800.0 PL=0
MOVL C01456 V=800.0 PL=0
MOVL C01457 V=800.0 PL=0
MOVL C01458 V=800.0 PL=0
MOVL C01459 V=800.0 PL=0
MOVL C01460 V=800.0 PL=0
MOVL C01461 V=800.0 PL=0
MOVL C01462 V=800.0 PL=0
MOVL C01463 V=800.0 PL=0
MOVL C01464 V=800.0 PL=0
MOVL C01465 V=800.0 PL=0
MOVL C01466 V=800.0 PL=0
MOVL C01467 V=800.0 PL=0
MOVL C01468 V=800.0 PL=0
MOVL C01469 V=800.0 PL=0
MOVL C01470 V=800.0 PL=0
MOVL C01471 V=800.0 PL=0
MOVL C01472 V=800.0 PL=0
MOVL C01473 V=800.0 PL=0
MOVL C01474 V=800.0 PL=0
MOVL C01475 V=800.0 PL=0
MOVL C01476 V=800.0 PL=0
MOVL C01477 V=800.0 PL=0
MOVL C01478 V=800.0 PL=0
MOVL C01479 V=800.0 PL=0
MOVL C01480 V=800.0 PL=0
MOVL C01481 V=800.0 PL=0
MOVL C01482 V=800.0 PL=0
MOVL C01483 V=800.0 PL=0
MOVL C01484 V=800.0 PL=0
MOVL C01485 V=800.0 PL=0
MOVL C01486 V=800.0 PL=0
MOVL C01487 V=800.0 PL=0
MOVL C01488 V=800.0 PL=0
MOVL C01489 V=800.0 PL=0
MOVL C01490 V=800.0 PL=0
MOVL C01491 V=800.0 PL=0
MOVL C01492 V=800.0 PL=0
MOVL C01493 V=800.0 PL=0
MOVL C01494 V=800.0 PL=0
MOVL C01495 V=800.0 PL=0
MOVL C01496 V=800.0 PL=0
MOVL C01497 V=800.0 PL=0
MOVL C01498 V=800.0 PL=0
MOVL C01499 V=800.0 PL=0
MOVL C01500 V=800.0 PL=0
MOVL C01501 V=800.0 PL=0
MOVL C01502 V=800.0 PL=0
MOVL C01503 V=800.0 PL=0
MOVL C01504 V=800.0 PL=0
MOVL C01505 V=800.0 PL=0
MOVL C01506 V=800.0 PL=0
MOVL C01507 V=800.0 PL=0
MOVL C01508 V=800.0 PL=0
MOVL C01509 V=800.0 PL=0
MOVL C01510 V=800.0 PL=0
MOVL C01511 V=800.0 PL=0
MOVL C01512 V=800.0 PL=0
MOVL C01513 V=800.0 PL=0
MOVL C01514 V=800.0 PL=0
MOVL C01515 V=800.0 PL=0
MOVL C01516 V=800.0 PL=0
MOVL C01517 V=800.0 PL=0
MOVL C01518 V=800.0 PL=0
MOVL C01519 V=800.0 PL=0
MOVL C01520 V=800.0 PL=0
MOVL C01521 V=800.0 PL=0
MOVL C01522 V=800.0 PL=0
MOVL C01523 V=800.0 PL=0
MOVL C01524 V=800.0 PL=0
MOVL C01525 V=800.0 PL=0
MOVL C01526 V=800.0 PL=0
MOVL C01527 V=800.0 PL=0
MOVL C01528 V=800.0 PL=0
MOVL C01529 V=800.0 PL=0
MOVL C01530 V=800.0 PL=0
MOVL C01531 V=800.0 PL=0
MOVL C01532 V=800.0 PL=0
MOVL C01533 V=800.0 PL=0
MOVL C01534 V=800.0 PL=0
MOVL C01535 V=800.0 PL=0
MOVL C01536 V=800.0 PL=0
MOVL C01537 V=800.0 PL=0
MOVL C01538 V=800.0 PL=0
MOVL C01539 V=800.0 PL=0
MOVL C01540 V=800.0 PL=0
MOVL C01541 V=800.0 PL=0
MOVL C01542 V=800.0 PL=0
MOVL C01543 V=800.0 PL=0
MOVL C01544 V=800.0 PL=0
MOVL C01545 V=800.0 PL=0
MOVL C01546 V=800.0 PL=0
MOVL C01547 V=800.0 PL=0
MOVL C01548 V=800.0 PL=0
MOVL C01549 V=800.0 PL=0
MOVL C01550 V=800.0 PL=0
MOVL C01551 V=800.0 PL=0
MOVL C01552 V=800.0 PL=0
MOVL C01553 V=800.0 PL=0
MOVL C01554 V=800.0 PL=0
MOVL C01555 V=800.0 PL=0
MOVL C01556 V=800.0 PL=0
MOVL C01557 V=800.0 PL=0
MOVL C01558 V=800.0 PL=0
MOVL C01559 V=800.0 PL=0
MOVL C01560 V=800.0 PL=0
MOVL C01561 V=800.0 PL=0
MOVL C01562 V=800.0 PL=0
MOVL C01563 V=800.0 PL=0
MOVL C01564 V=800.0 PL=0
MOVL C01565 V=800.0 PL=0
MOVL C01566 V=800.0 PL=0
MOVL C01567 V=800.0 PL=0
MOVL C01568 V=800.0 PL=0
MOVL C01569 V=800.0 PL=0
MOVL C01570 V=800.0 PL=0
MOVL C01571 V=800.0 PL=0
MOVL C01572 V=800.0 PL=0
MOVL C01573 V=800.0 PL=0
MOVL C01574 V=800.0 PL=0
MOVL C01575 V=800.0 PL=0
MOVL C01576 V=800.0 PL=0
MOVL C01577 V=800.0 PL=0
MOVL C01578 V=800.0 PL=0
MOVL C01579 V=800.0 PL=0
MOVL C01580 V=800.0 PL=0
MOVL C01581 V=800.0 PL=0
MOVL C01582 V=800.0 PL=0
MOVL C01583 V=800.0 PL=0
MOVL C01584 V=800.0 PL=0
MOVL C01585 V=800.0 PL=0
MOVL C01586 V=800.0 PL=0
MOVL C01587 V=800.0 PL=0
MOVL C01588 V=800.0 PL=0
MOVL C01589 V=800.0 PL=0
MOVL C01590 V=800.0 PL=0
MOVL C01591 V=800.0 PL=0
MOVL C01592 V=800.0 PL=0
MOVL C01593 V=800.0 PL=0
MOVL C01594 V=800.0 PL=0
MOVL C01595 V=800.0 PL=0
MOVL C01596 V=800.0 PL=0
MOVL C01597 V=800.0 PL=0
MOVL C01598 V=800.0 PL=0
MOVL C01599 V=800.0 PL=0
MOVL C01600 V=800.0 PL=0
MOVL C01601 V=800.0 PL=0
MOVL C01602 V=800.0 PL=0
MOVL C01603 V=800.0 PL=0
MOVL C01604 V=800.0 PL=0
MOVL C01605 V=800.0 PL=0
MOVL C01606 V=800.0 PL=0
MOVL C01607 V=800.0 PL=0
MOVL C01608 V=800.0 PL=0
MOVL C01609 V=800.0 PL=0
MOVL C01610 V=800.0 PL=0
MOVL C01611 V=800.0 PL=0
MOVL C01612 V=800.0 PL=0
MOVL C01613 V=800.0 PL=0
MOVL C01614 V=800.0 PL=0
MOVL C01615 V=800.0 PL=0
MOVL C01616 V=800.0 PL=0
MOVL C01617 V=800.0 PL=0
MOVL C01618 V=800.0 PL=0
MOVL C01619 V=800.0 PL=0
MOVL C01620 V=800.0 PL=0
MOVL C01621 V=800.0 PL=0
MOVL C01622 V=800.0 PL=0
MOVL C01623 V=800.0 PL=0
MOVL C01624 V=800.0 PL=0
MOVL C01625 V=800.0 PL=0
MOVL C01626 V=800.0 PL=0
MOVL C01627 V=800.0 PL=0
MOVL C01628 V=800.0 PL=0
MOVL C01629 V=800.0 PL=0
MOVL C01630 V=800.0 PL=0
MOVL C01631 V=800.0 PL=0
MOVL C01632 V=800.0 PL=0
MOVL C01633 V=800.0 PL=0
MOVL C01634 V=800.0 PL=0
MOVL C01635 V=800.0 PL=0
MOVL C01636 V=800.0 PL=0
MOVL C01637 V=800.0 PL=0
MOVL C01638 V=800.0 PL=0
MOVL C01639 V=800.0 PL=0
MOVL C01640 V=800.0 PL=0
MOVL C01641 V=800.0 PL=0
MOVL C01642 V=800.0 PL=0
MOVL C01643 V=800.0 PL=0
MOVL C01644 V=800.0 PL=0
MOVL C01645 V=800.0 PL=0
MOVL C01646 V=800.0 PL=0
MOVL C01647 V=800.0 PL=0
MOVL C01648 V=800.0 PL=0
MOVL C01649 V=800.0 PL=0
MOVL C01650 V=800.0 PL=0
MOVL C01651 V=800.0 PL=0
MOVL C01652 V=800.0 PL=0
MOVL C01653 V=800.0 PL=0
MOVL C01654 V=800.0 PL=0
MOVL C01655 V=800.0 PL=0
MOVL C01656 V=800.0 PL=0
MOVL C01657 V=800.0 PL=0
MOVL C01658 V=800.0 PL=0
MOVL C01659 V=800.0 PL=0
MOVL C01660 V=800.0 PL=0
MOVL C01661 V=800.0 PL=0
MOVL C01662 V=800.0 PL=0
MOVL C01663 V=800.0 PL=0
MOVL C01664 V=800.0 PL=0
MOVL C01665 V=800.0 PL=0
MOVL C01666 V=800.0 PL=0
MOVL C01667 V=800.0 PL=0
MOVL C01668 V=800.0 PL=0
MOVL C01669 V=800.0 PL=0
MOVL C01670 V=800.0 PL=0
MOVL C01671 V=800.0 PL=0
MOVL C01672 V=800.0 PL=0
MOVL C01673 V=800.0 PL=0
MOVL C01674 V=800.0 PL=0
MOVL C01675 V=800.0 PL=0
MOVL C01676 V=800.0 PL=0
MOVL C01677 V=800.0 PL=0
MOVL C01678 V=800.0 PL=0
MOVL C01679 V=800.0 PL=0
MOVL C01680 V=800.0 PL=0
MOVL C01681 V=800.0 PL=0
MOVL C01682 V=800.0 PL=0
MOVL C01683 V=800.0 PL=0
MOVL C01684 V=800.0 PL=0
MOVL C01685 V=800.0 PL=0
MOVL C01686 V=800.0 PL=0
MOVL C01687 V=800.0 PL=0
MOVL C01688 V=800.0 PL=0
MOVL C01689 V=800.0 PL=0
MOVL C01690 V=800.0 PL=0
MOVL C01691 V=800.0 PL=0
MOVL C01692 V=800.0 PL=0
MOVL C01693 V=800.0 PL=0
MOVL C01694 V=800.0 PL=0
MOVL C01695 V=800.0 PL=0
MOVL C01696 V=800.0 PL=0
MOVL C01697 V=800.0 PL=0
MOVL C01698 V=800.0 PL=0
MOVL C01699 V=800.0 PL=0
MOVL C01700 V=800.0 PL=0
MOVL C01701 V=800.0 PL=0
MOVL C01702 V=800.0 PL=0
MOVL C01703 V=800.0 PL=0
MOVL C01704 V=800.0 PL=0
MOVL C01705 V=800.0 PL=0
MOVL C01706 V=800.0 PL=0
MOVL C01707 V=800.0 PL=0
MOVL C01708 V=800.0 PL=0
MOVL C01709 V=800.0 PL=0
MOVL C01710 V=800.0 PL=0
MOVL C01711 V=800.0 PL=0
MOVL C01712 V=800.0 PL=0
MOVL C01713 V=800.0 PL=0
MOVL C01714 V=800.0 PL=0
MOVL C01715 V=800.0 PL=0
MOVL C01716 V=800.0 PL=0
MOVL C01717 V=800.0 PL=0
MOVL C01718 V=800.0 PL=0
MOVL C01719 V=800.0 PL=0
MOVL C01720 V=800.0 PL=0
MOVL C01721 V=800.0 PL=0
MOVL C01722 V=800.0 PL=0
MOVL C01723 V=800.0 PL=0
MOVL C01724 V=800.0 PL=0
MOVL C01725 V=800.0 PL=0
MOVL C01726 V=800.0 PL=0
MOVL C01727 V=800.0 PL=0
MOVL C01728 V=800.0 PL=0
MOVL C01729 V=800.0 PL=0
MOVL C01730 V=800.0 PL=0
MOVL C01731 V=800.0 PL=0
MOVL C01732 V=800.0 PL=0
MOVL C01733 V=800.0 PL=0
MOVL C01734 V=800.0 PL=0
MOVL C01735 V=800.0 PL=0
MOVL C01736 V=800.0 PL=0
MOVL C01737 V=800.0 PL=0
MOVL C01738 V=800.0 PL=0
MOVL C01739 V=800.0 PL=0
MOVL C01740 V=800.0 PL=0
MOVL C01741 V=800.0 PL=0
MOVL C01742 V=800.0 PL=0
MOVL C01743 V=800.0 PL=0
MOVL C01744 V=800.0 PL=0
MOVL C01745 V=800.0 PL=0
MOVL C01746 V=800.0 PL=0
MOVL C01747 V=800.0 PL=0
MOVL C01748 V=800.0 PL=0
MOVL C01749 V=800.0 PL=0
MOVL C01750 V=800.0 PL=0
MOVL C01751 V=800.0 PL=0
MOVL C01752 V=800.0 PL=0
MOVL C01753 V=800.0 PL=0
MOVL C01754 V=800.0 PL=0
MOVL C01755 V=800.0 PL=0
MOVL C01756 V=800.0 PL=0
MOVL C01757 V=800.0 PL=0
MOVL C01758 V=800.0 PL=0
MOVL C01759 V=800.0 PL=0
MOVL C01760 V=800.0 PL=0
MOVL C01761 V=800.0 PL=0
MOVL C01762 V=800.0 PL=0
MOVL C01763 V=800.0 PL=0
MOVL C01764 V=800.0 PL=0
MOVL C01765 V=800.0 PL=0
MOVL C01766 V=800.0 PL=0
MOVL C01767 V=800.0 PL=0
MOVL C01768 V=800.0 PL=0
MOVL C01769 V=800.0 PL=0
MOVL C01770 V=800.0 PL=0
MOVL C01771 V=800.0 PL=0
MOVL C01772 V=800.0 PL=0
MOVL C01773 V=800.0 PL=0
MOVL C01774 V=800.0 PL=0
MOVL C01775 V=800.0 PL=0
MOVL C01776 V=800.0 PL=0
MOVL C01777 V=800.0 PL=0
MOVL C01778 V=800.0 PL=0
MOVL C01779 V=800.0 PL=0
MOVL C01780 V=800.0 PL=0
MOVL C01781 V=800.0 PL=0
MOVL C01782 V=800.0 PL=0
MOVL C01783 V=800.0 PL=0
MOVL C01784 V=800.0 PL=0
MOVL C01785 V=800.0 PL=0
MOVL C01786 V=800.0 PL=0
MOVL C01787 V=800.0 PL=0
MOVL C01788 V=800.0 PL=0
MOVL C01789 V=800.0 PL=0
MOVL C01790 V=800.0 PL=0
MOVL C01791 V=800.0 PL=0
MOVL C01792 V=800.0 PL=0
MOVL C01793 V=800.0 PL=0
MOVL C01794 V=800.0 PL=0
MOVL C01795 V=800.0 PL=0
MOVL C01796 V=800.0 PL=0
MOVL C01797 V=800.0 PL=0
MOVL C01798 V=800.0 PL=0
MOVL C01799 V=800.0 PL=0
MOVL C01800 V=800.0 PL=0
MOVL C01801 V=800.0 PL=0
MOVL C01802 V=800.0 PL=0
MOVL C01803 V=800.0 PL=0
MOVL C01804 V=800.0 PL=0
MOVL C01805 V=800.0 PL=0
MOVL C01806 V=800.0 PL=0
MOVL C01807 V=800.0 PL=0
MOVL C01808 V=800.0 PL=0
MOVL C01809 V=800.0 PL=0
MOVL C01810 V=800.0 PL=0
MOVL C01811 V=800.0 PL=0
MOVL C01812 V=800.0 PL=0
MOVL C01813 V=800.0 PL=0
MOVL C01814 V=800.0 PL=0
MOVL C01815 V=800.0 PL=0
MOVL C01816 V=800.0 PL=0
MOVL C01817 V=800.0 PL=0
MOVL C01818 V=800.0 PL=0
MOVL C01819 V=800.0 PL=0
MOVL C01820 V=800.0 PL=0
MOVL C01821 V=800.0 PL=0
MOVL C01822 V=800.0 PL=0
MOVL C01823 V=800.0 PL=0
MOVL C01824 V=800.0 PL=0
MOVL C01825 V=800.0 PL=0
MOVL C01826 V=800.0 PL=0
MOVL C01827 V=800.0 PL=0
MOVL C01828 V=800.0 PL=0
MOVL C01829 V=800.0 PL=0
MOVL C01830 V=800.0 PL=0
MOVL C01831 V=800.0 PL=0
MOVL C01832 V=800.0 PL=0
MOVL C01833 V=800.0 PL=0
MOVL C01834 V=800.0 PL=0
MOVL C01835 V=800.0 PL=0
MOVL C01836 V=800.0 PL=0
MOVL C01837 V=800.0 PL=0
MOVL C01838 V=800.0 PL=0
MOVL C01839 V=800.0 PL=0
MOVL C01840 V=800.0 PL=0
MOVL C01841 V=800.0 PL=0
MOVL C01842 V=800.0 PL=0
MOVL C01843 V=800.0 PL=0
MOVL C01844 V=800.0 PL=0
MOVL C01845 V=800.0 PL=0
MOVL C01846 V=800.0 PL=0
MOVL C01847 V=800.0 PL=0
MOVL C01848 V=800.0 PL=0
MOVL C01849 V=800.0 PL=0
MOVL C01850 V=800.0 PL=0
MOVL C01851 V=800.0 PL=0
MOVL C01852 V=800.0 PL=0
MOVL C01853 V=800.0 PL=0
MOVL C01854 V=800.0 PL=0
MOVL C01855 V=800.0 PL=0
MOVL C01856 V=800.0 PL=0
MOVL C01857 V=800.0 PL=0
MOVL C01858 V=800.0 PL=0
MOVL C01859 V=800.0 PL=0
MOVL C01860 V=800.0 PL=0
MOVL C01861 V=800.0 PL=0
MOVL C01862 V=800.0 PL=0
MOVL C01863 V=800.0 PL=0
MOVL C01864 V=800.0 PL=0
MOVL C01865 V=800.0 PL=0
MOVL C01866 V=800.0 PL=0
MOVL C01867 V=800.0 PL=0
MOVL C01868 V=800.0 PL=0
MOVL C01869 V=800.0 PL=0
MOVL C01870 V=800.0 PL=0
MOVL C01871 V=800.0 PL=0
MOVL C01872 V=800.0 PL=0
MOVL C01873 V=800.0 PL=0
MOVL C01874 V=800.0 PL=0
MOVL C01875 V=800.0 PL=0
MOVL C01876 V=800.0 PL=0
MOVL C01877 V=800.0 PL=0
MOVL C01878 V=800.0 PL=0
MOVL C01879 V=800.0 PL=0
MOVL C01880 V=800.0 PL=0
MOVL C01881 V=800.0 PL=0
MOVL C01882 V=800.0 PL=0
MOVL C01883 V=800.0 PL=0
MOVL C01884 V=800.0 PL=0
MOVL C01885 V=800.0 PL=0
MOVL C01886 V=800.0 PL=0
MOVL C01887 V=800.0 PL=0
MOVL C01888 V=800.0 PL=0
MOVL C01889 V=800.0 PL=0
MOVL C01890 V=800.0 PL=0
MOVL C01891 V=800.0 PL=0
MOVL C01892 V=800.0 PL=0
MOVL C01893 V=800.0 PL=0
MOVL C01894 V=800.0 PL=0
MOVL C01895 V=800.0 PL=0
MOVL C01896 V=800.0 PL=0
MOVL C01897 V=800.0 PL=0
MOVL C01898 V=800.0 PL=0
MOVL C01899 V=800.0 PL=0
MOVL C01900 V=800.0 PL=0
MOVL C01901 V=800.0 PL=0
MOVL C01902 V=800.0 PL=0
MOVL C01903 V=800.0 PL=0
MOVL C01904 V=800.0 PL=0
MOVL C01905 V=800.0 PL=0
MOVL C01906 V=800.0 PL=0
MOVL C01907 V=800.0 PL=0
MOVL C01908 V=800.0 PL=0
MOVL C01909 V=800.0 PL=0
MOVL C01910 V=800.0 PL=0
MOVL C01911 V=800.0 PL=0
MOVL C01912 V=800.0 PL=0
MOVL C01913 V=800.0 PL=0
MOVL C01914 V=800.0 PL=0
MOVL C01915 V=800.0 PL=0
MOVL C01916 V=800.0 PL=0
MOVL C01917 V=800.0 PL=0
MOVL C01918 V=800.0 PL=0
MOVL C01919 V=800.0 PL=0
MOVL C01920 V=800.0 PL=0
MOVL C01921 V=800.0 PL=0
MOVL C01922 V=800.0 PL=0
MOVL C01923 V=800.0 PL=0
MOVL C01924 V=800.0 PL=0
MOVL C01925 V=800.0 PL=0
MOVL C01926 V=800.0 PL=0
MOVL C01927 V=800.0 PL=0
MOVL C01928 V=800.0 PL=0
MOVL C01929 V=800.0 PL=0
MOVL C01930 V=800.0 PL=0
MOVL C01931 V=800.0 PL=0
MOVL C01932 V=800.0 PL=0
MOVL C01933 V=800.0 PL=0
MOVL C01934 V=800.0 PL=0
MOVL C01935 V=800.0 PL=0
MOVL C01936 V=800.0 PL=0
MOVL C01937 V=800.0 PL=0
MOVL C01938 V=800.0 PL=0
MOVL C01939 V=800.0 PL=0
MOVL C01940 V=800.0 PL=0
MOVL C01941 V=800.0 PL=0
MOVL C01942 V=800.0 PL=0
MOVL C01943 V=800.0 PL=0
MOVL C01944 V=800.0 PL=0
MOVL C01945 V=800.0 PL=0
MOVL C01946 V=800.0 PL=0
MOVL C01947 V=800.0 PL=0
MOVL C01948 V=800.0 PL=0
MOVL C01949 V=800.0 PL=0
MOVL C01950 V=800.0 PL=0
MOVL C01951 V=800.0 PL=0
MOVL C01952 V=800.0 PL=0
MOVL C01953 V=800.0 PL=0
MOVL C01954 V=800.0 PL=0
MOVL C01955 V=800.0 PL=0
MOVL C01956 V=800.0 PL=0
MOVL C01957 V=800.0 PL=0
MOVL C01958 V=800.0 PL=0
MOVL C01959 V=800.0 PL=0
MOVL C01960 V=800.0 PL=0
MOVL C01961 V=800.0 PL=0
MOVL C01962 V=800.0 PL=0
MOVL C01963 V=800.0 PL=0
MOVL C01964 V=800.0 PL=0
MOVL C01965 V=800.0 PL=0
MOVL C01966 V=800.0 PL=0
MOVL C01967 V=800.0 PL=0
MOVL C01968 V=800.0 PL=0
MOVL C01969 V=800.0 PL=0
MOVL C01970 V=800.0 PL=0
MOVL C01971 V=800.0 PL=0
MOVL C01972 V=800.0 PL=0
MOVL C01973 V=800.0 PL=0
MOVL C01974 V=800.0 PL=0
MOVL C01975 V=800.0 PL=0
MOVL C01976 V=800.0 PL=0
MOVL C01977 V=800.0 PL=0
MOVL C01978 V=800.0 PL=0
MOVL C01979 V=800.0 PL=0
MOVL C01980 V=800.0 PL=0
MOVL C01981 V=800.0 PL=0
MOVL C01982 V=800.0 PL=0
MOVL C01983 V=800.0 PL=0
MOVL C01984 V=800.0 PL=0
MOVL C01985 V=800.0 PL=0
MOVL C01986 V=800.0 PL=0
MOVL C01987 V=800.0 PL=0
MOVL C01988 V=800.0 PL=0
MOVL C01989 V=800.0 PL=0
MOVL C01990 V=800.0 PL=0
MOVL C01991 V=800.0 PL=0
MOVL C01992 V=800.0 PL=0
MOVL C01993 V=800.0 PL=0
MOVL C01994 V=800.0 PL=0
MOVL C01995 V=800.0 PL=0
MOVL C01996 V=800.0 PL=0
MOVL C01997 V=800.0 PL=0
MOVL C01998 V=800.0 PL=0
MOVL C01999 V=800.0 PL=0
MOVL C02000 V=800.0 PL=0
MOVL C02001 V=800.0 PL=0
MOVL C02002 V=800.0 PL=0
MOVL C02003 V=800.0 PL=0
MOVL C02004 V=800.0 PL=0
MOVL C02005 V=800.0 PL=0
MOVL C02006 V=800.0 PL=0
MOVL C02007 V=800.0 PL=0
MOVL C02008 V=800.0 PL=0
MOVL C02009 V=800.0 PL=0
MOVL C02010 V=800.0 PL=0
MOVL C02011 V=800.0 PL=0
MOVL C02012 V=800.0 PL=0
MOVL C02013 V=800.0 PL=0
MOVL C02014 V=800.0 PL=0
MOVL C02015 V=800.0 PL=0
MOVL C02016 V=800.0 PL=0
MOVL C02017 V=800.0 PL=0
MOVL C02018 V=800.0 PL=0
MOVL C02019 V=800.0 PL=0
MOVL C02020 V=800.0 PL=0
MOVL C02021 V=800.0 PL=0
MOVL C02022 V=800.0 PL=0
MOVL C02023 V=800.0 PL=0
MOVL C02024 V=800.0 PL=0
MOVL C02025 V=800.0 PL=0
MOVL C02026 V=800.0 PL=0
MOVL C02027 V=800.0 PL=0
MOVL C02028 V=800.0 PL=0
MOVL C02029 V=800.0 PL=0
MOVL C02030 V=800.0 PL=0
MOVL C02031 V=800.0 PL=0
MOVL C02032 V=800.0 PL=0
MOVL C02033 V=800.0 PL=0
MOVL C02034 V=800.0 PL=0
MOVL C02035 V=800.0 PL=0
MOVL C02036 V=800.0 PL=0
MOVL C02037 V=800.0 PL=0
MOVL C02038 V=800.0 PL=0
MOVL C02039 V=800.0 PL=0
MOVL C02040 V=800.0 PL=0
MOVL C02041 V=800.0 PL=0
MOVL C02042 V=800.0 PL=0
MOVL C02043 V=800.0 PL=0
MOVL C02044 V=800.0 PL=0
MOVL C02045 V=800.0 PL=0
MOVL C02046 V=800.0 PL=0
MOVL C02047 V=800.0 PL=0
MOVL C02048 V=800.0 PL=0
MOVL C02049 V=800.0 PL=0
